Universal Robots URScript: faichun_snake3.script

def faichun_snake3():
  set_tool_communication(True, 1000000, 2, 1, 1.5, 3.5)
  set_tool_output_mode(0)
  set_tool_digital_output_mode(0, 1)
  set_tool_digital_output_mode(1, 1)
  set_tool_voltage(24)
  step_count_e741a7f4_0b30_46a8_b996_4636aff9ce90 = 0.0
  thread Step_Counter_Thread_bd4b55fe_d110_495a_a627_b98bcdc962aa():
    while (True):
      step_count_e741a7f4_0b30_46a8_b996_4636aff9ce90 = step_count_e741a7f4_0b30_46a8_b996_4636aff9ce90 + 1.0
      sync()
    end
  end
  run Step_Counter_Thread_bd4b55fe_d110_495a_a627_b98bcdc962aa()
  set_gravity([0.0, 0.0, 9.82])
  set_tcp(p[0.0,0.0,0.0,0.0,0.0,0.0])
  set_standard_analog_input_domain(0, 1)
  set_standard_analog_input_domain(1, 1)
  set_tool_analog_input_domain(0, 1)
  set_tool_analog_input_domain(1, 1)
  set_analog_outputdomain(0, 0)
  set_analog_outputdomain(1, 0)
  set_input_actions_to_default()
  set_safety_mode_transition_hardness(1)
  set_target_payload(1.070000, [0.002000, 0.003000, 0.057000], [0.001723, 0.001723, 0.001723, 0.000000, 0.000000, 0.000000])
  global B1empty=False
  global A2Empty=0
  global A1Empty=0
  global B2Empty=False
  global pallet_step=0
  global bright_box=0
  global Pallet_1_cnt=2
  global dark_boxes=0
  global Point_1=p[0.6913645118948067,-0.12399382748223003,0.49223711947071,-1.2983729986843258,1.1259514972191385,-1.2203503861141718]
  # begin: URCap Installation Node
  #   Source: External Control, 1.0.5, FZI Research Center for Information Technology
  #   Type: External Control
  # end: URCap Installation Node
  # begin: URCap Installation Node
  #   Source: OnRobot, 6.2.0, OnRobot A/S
  #   Type: OnRobot Setup
  sleep(1)
  if (False):
  end
  ON_CONN_SHIFT_BOOL = 64
  ON_CONN_SHIFT_INT = 24
  ON_CONN_SHIFT_FLOAT = 24
  ON_CONN_REG_SUM_BOOL = 0
  ON_CONN_REG_SUM_INT = 1
  ON_CONN_REG_SUM_FLOAT = 0
  ON_TOOL_SHIFT_BOOL = 64
  ON_TOOL_SHIFT_INT = 25
  ON_TOOL_SHIFT_FLOAT = 24
  ON_TOOL_SHIFT_BOOL_ARR = [64, 64, 64]
  ON_TOOL_SHIFT_INT_ARR = [25, 25, 25]
  ON_TOOL_SHIFT_FLOAT_ARR = [24, 24, 24]
  ON_TOOL_REG_SUM_BOOL = 0
  ON_TOOL_REG_SUM_INT = 0
  ON_TOOL_REG_SUM_FLOAT = 0
  ON_REGISTERS_SPEEDL_FLOAT = 0
  ON_REG_USE_TOOL = False
  ON_DI_SINGLE = 0
  ON_DI_PRIMARY = 1
  ON_DI_SECONDARY = 2
  ON_DI_DUAL = 3
  on_robot_type = 10
  on_robot_cycle = 2.0
  on_conn_ip = "localhost"
  on_tool_ip = "localhost"
  on_device_socket_port = 51234
  on_conn_xmlrpc = rpc_factory("xmlrpc", "http://localhost:41414")
  on_tool_xmlrpc = rpc_factory("xmlrpc", "http://localhost:41414")
  on_RPC = rpc_factory("xmlrpc", "http://127.0.0.1:31416")
  ON_DEBUG_LOG = False
  on_isMetric = True
  on_toolConnector = True
  on_ioqc = False
  on_dual = False
  on_computebox = False
  on_devices = 0
  on_gripper = [False, False, False]
  on_custom_tcp_id = "none"
  on_custom_tcp_enabled = False
  speedlTime = 0.001
  on_ft = False
  #======    OnRobot Globals    ======#

  ON_MATH_PI=3.141593
  ON_ZEROPOSE=p[0.0,0.0,0.0,0.0,0.0,0.0]
  ON_ZEROFRAME=p[0.0,0.0,0.0,0.0,0.0,0.0]
  ON_ZERO3D=[0.0,0.0,0.0]
  ON_ZERO6D=[0.0,0.0,0.0,0.0,0.0,0.0]
  ON_ZERO8D=[0.0,0.0,0.0,0.0,0.0,0.0,0.0,0.0]
  ON_FALSE3D=[False,False,False]
  ON_FALSE6D=[False,False,False,False,False,False]
  ON_FALSE8D=[False,False,False,False,False,False,False,False]
  global on_return=0
  on_speedL=ON_ZERO6D
  on_speedBase=ON_ZERO6D
  on_speedVect=ON_ZERO6D
  on_speedExtra=ON_ZERO6D
  on_speedCB=ON_ZERO6D
  on_speedGecko=ON_ZERO6D
  on_RTDE_error=0
  on_RTDE_tool_error=0
  on_dataProcess_thrd=0
  ON_DEVICE_ID_MISSING=0
  ON_INIT_WATCHDOG_HZ=5
  ON_INIT_TIMEOUT=2000
  on_robot_TCP_offset=ON_ZEROFRAME
  on_tcp_offset_actual=ON_ZEROFRAME
  on_cog_actual=ON_ZEROFRAME
  on_mass_actual=0.0
  on_robot_mount=[0.0,0.0]

  #======    End of OnRobot Globals    ======#
  #======    OnRobot Interface Messages    ======#

  on_devices_primary_log="OnRobot Devices"
  on_devices_secondary_log="OnRobot Secondary Device"
  on_program_halted="<br>Program halted."
  on_device_error_title="OnRobot - Device error"
  on_install_error="OnRobot Setup is not correct.<br>Check the status in the OnRobot Setup page in the Installation Tab.<br>Program halted."
  on_device_missing="No device connected.<br>Program halted."
  cb_device_missing="No OnRobot Compute Box connected.<br>Program halted."
  ft_device_missing="No OnRobot FT sensor or license detected.<br>Program halted."
  hex_device_missing="No HEX sensor connected.<br>Program halted."
  rg2ft_device_missing="No RG2-FT gripper connected.<br>Program halted."
  rg_device_missing="No RG gripper connected.<br>Program halted."
  vg_device_missing="No VG gripper connected.<br>Program halted."
  gg_device_missing="No Gecko Gripper connected.<br>Program halted."
  sg_device_missing="No Soft Gripper connected.<br>Program halted."
  tfg_device_missing="No 3FG gripper connected.<br>Program halted."
  sdr_device_missing="No OnRobot Sander connected.<br>Program halted."
  twofg_device_missing="No 2FG gripper connected.<br>Program halted."
  vgp_device_missing="No VGP gripper connected.<br>Program halted."
  mg_device_missing="No Magnetic Gripper connected.<br>Program halted."
  fgp_device_missing="No 2FGP20 Gripper connected.<br>Program halted."
  eyes_device_missing="No OnRobot Eyes connected.<br>Program halted."
  on_xmlrpc_start_ip="Connecting to OnRobot XML-RPC Server:"
  on_java_comm_error_textmsg_title="OnRobot - Communication error:"
  on_java_comm_controlsocket_open_error="Socket 'javaSocket' opening was unsuccessful."
  on_java_comm_error_title="OnRobot - Communication error"
  on_java_comm_socket_open_error="Establishing connection with the URCap was timed out.<br>Check the status in the OnRobot Setup page in the Installation Tab.<br>Program halted."
  on_rtde_feed_error_textmsg_title="OnRobot - RTDE error:"
  on_rtde_feed_error="RTDE feed error. OnRobot device count mismatch.<br>Program halted."
  on_rtde_feed_tool_error="Tool RTDE feed error. OnRobot device count mismatch.<br>Program halted."
  on_rtde_feed_open_error_textmsg="Socket 'rtdeFeed' opening was unsuccessful."
  on_rtde_feed_error_title="OnRobot - RTDE error"
  on_rtde_feed_count_error="Invalid RTDE offset setup detected. Please check RTDE Offsets at the OnRobot Setup page in the Installation Tab.<br>Program halted."
  on_rtde_feed_open_error="Establishing connection with the devices was timed out.<br>Ensure that the OnRobot devices are operational, and check the status in the OnRobot Setup page in the Installation Tab."

  #======    End of OnRobot Interface Messages    ======#
  #======    OnRobot Interface    ======#

  on_portopened_javaSocket=False
  on_rtde_feed_opened=False
  on_dataProcess_running=False
  def on_missing():
  popup(on_device_missing,title=on_device_error_title,error=True,blocking=False)
  halt
  end
  def cb_missing():
  popup(cb_device_missing,title=on_device_error_title,error=True,blocking=False)
  halt
  end
  def ft_missing():
  popup(ft_device_missing,title=on_device_error_title,error=True,blocking=False)
  halt
  end
  def hex_missing():
  popup(hex_device_missing,title=on_device_error_title,error=True,blocking=False)
  halt
  end
  def rg2ft_missing():
  popup(rg2ft_device_missing,title=on_device_error_title,error=True,blocking=False)
  halt
  end
  def rg_missing():
  popup(rg_device_missing,title=on_device_error_title,error=True,blocking=False)
  halt
  end
  def vg_missing():
  popup(vg_device_missing,title=on_device_error_title,error=True,blocking=False)
  halt
  end
  def gg_missing():
  popup(gg_device_missing,title=on_device_error_title,error=True,blocking=False)
  halt
  end
  def sg_missing():
  popup(sg_device_missing,title=on_device_error_title,error=True,blocking=False)
  halt
  end
  def tfg_missing():
  popup(tfg_device_missing,title=on_device_error_title,error=True,blocking=False)
  halt
  end
  def sdr_missing():
  popup(sdr_device_missing,title=on_device_error_title,error=True,blocking=False)
  halt
  end
  def twofg_missing():
  popup(twofg_device_missing,title=on_device_error_title,error=True,blocking=False)
  halt
  end
  def vgp_missing():
  popup(vgp_device_missing,title=on_device_error_title,error=True,blocking=False)
  halt
  end
  def mg_missing():
  popup(mg_device_missing,title=on_device_error_title,error=True,blocking=False)
  halt
  end
  def fgp_missing():
  popup(fgp_device_missing,title=on_device_error_title,error=True,blocking=False)
  halt
  end
  def eyes_missing():
  popup(eyes_device_missing,title=on_device_error_title,error=True,blocking=False)
  halt
  end
  def on_portclose_javaSocket():
  socket_close("javaSocket")
  on_portopened_javaSocket=False
  end
  def on_portopen_javaSocket():
  on_portclose_javaSocket()
  on_portopened_javaSocket=socket_open("127.0.0.1",44005,"javaSocket")
  if not on_portopened_javaSocket:
  textmsg(on_java_comm_error_textmsg_title,on_java_comm_controlsocket_open_error)
  popup(on_java_comm_socket_open_error,title=on_java_comm_error_title,error=True,blocking=False)
  halt
  end
  end
  on_conn_rtde_feed_name="rtdeFeedConn"
  on_tool_rtde_feed_name="rtdeFeedTool"
  def on_rtde_feed_close(rtdeFeedName):
  socket_close(rtdeFeedName)
  on_rtde_feed_opened=False
  end
  def on_rtde_feed_open(deviceIP,rtdeFeedName,regStart,regSum,regSpeedl):
  on_rtde_feed_close(rtdeFeedName)
  if((regStart[0]+regSum[0])>128)or((regStart[1]+regSum[1])>48)or((regStart[2]+regSum[2])>48):
  popup(on_rtde_feed_count_error,title=on_rtde_feed_error_title,error=True,blocking=False)
  textmsg(str_cat("RegStart: ",regStart),str_cat("  -  RegSum: ",regSum))
  halt
  end
  on_rtde_feed_opened=socket_open(deviceIP,on_device_socket_port,rtdeFeedName)
  if not on_rtde_feed_opened:
  on_rtde_feed_opened=socket_open(deviceIP,on_device_socket_port,rtdeFeedName)
  end
  if not on_rtde_feed_opened:
  textmsg(on_rtde_feed_error_textmsg_title,on_rtde_feed_open_error_textmsg)
  popup(on_rtde_feed_open_error,title=on_rtde_feed_error_title,error=True,blocking=False)
  halt
  end
  socket_send_int(regStart[0],rtdeFeedName)
  socket_send_int(regSum[0],rtdeFeedName)
  socket_send_int(regStart[1],rtdeFeedName)
  socket_send_int(regSum[1],rtdeFeedName)
  socket_send_int(regStart[2],rtdeFeedName)
  socket_send_int(regSum[2],rtdeFeedName)
  socket_send_int(regSpeedl,rtdeFeedName)
  socket_send_int(on_devices,rtdeFeedName)
  end
  def on_dataRead():
  enter_critical
  on_RTDE_error=read_input_integer_register(ON_CONN_SHIFT_INT)
  if(ON_REG_USE_TOOL):
  on_RTDE_tool_error=read_input_integer_register(ON_TOOL_SHIFT_INT_ARR[0])
  end
  exit_critical
  end
  def on_set_rtde_watchdog(updateHz=ON_INIT_WATCHDOG_HZ):
  local effect="stop"
  if(updateHz<1):
  effect="ignore"
  end
  watchdog_conn_reg_str=str_cat("input_int_register_",ON_CONN_SHIFT_INT)
  rtde_set_watchdog(watchdog_conn_reg_str,updateHz,effect)
  if(ON_REG_USE_TOOL):
  watchdog_tool_reg_str=str_cat("input_int_register_",ON_TOOL_SHIFT_INT_ARR[0])
  rtde_set_watchdog(watchdog_tool_reg_str,updateHz,effect)
  end
  if ON_DEBUG_LOG:
  local update_str=str_cat(" "+effect+" watchdog set to [Hz]: ",updateHz)
  textmsg(watchdog_conn_reg_str,update_str)
  if(ON_REG_USE_TOOL):
  local update_str=str_cat(" "+effect+" watchdog set to [Hz]: ",updateHz)
  textmsg(watchdog_tool_reg_str,update_str)
  end
  end
  end
  def on_speedCB_get():
  return[on_speedCB[0],on_speedCB[1],on_speedCB[2],on_speedCB[3],on_speedCB[4],on_speedCB[5]]
  end
  def on_speedGecko_get():
  local speedExtra=ON_ZERO6D
  if on_speedl_for_gecko:
  speedExtra=[on_speedGecko[0],on_speedGecko[1],on_speedGecko[2],on_speedGecko[3],on_speedGecko[4],on_speedGecko[5]]
  end
  return speedExtra
  end
  def on_speedGecko_set(speedGecko):
  on_speedGecko=[speedGecko[0],speedGecko[1],speedGecko[2],speedGecko[3],speedGecko[4],speedGecko[5]]
  end
  thread on_dataProcess_thread():
  if ON_DEBUG_LOG:
  textmsg("Starting on_dataRead thread")
  end
  local error=False
  on_dataProcess_running=True
  sync()
  while on_dataProcess_running:
  sync()
  on_dataRead()
  error=on_error((on_RTDE_error<0),on_rtde_feed_error,on_rtde_feed_error_title,error)
  error=on_error((ON_REG_USE_TOOL and(on_RTDE_tool_error<0)),on_rtde_feed_tool_error,on_rtde_feed_error_title,error)
  on_dataProcess_running=not error
  end
  if error:
  halt
  end
  if ON_DEBUG_LOG:
  textmsg("Stopping on_dataRead thread")
  end
  end
  thread on_set_watchdog_thread():
  sleep(2)
  on_set_rtde_watchdog(updateHz=ON_INIT_WATCHDOG_HZ)
  sleep(1/ON_INIT_WATCHDOG_HZ)
  on_dataProcess_running=False
  kill on_dataProcess_thrd
  end

  #======    End of OnRobot Interface    ======#
  #======    OnRobot QC Setup Tool Connector    ======#

  def tc_setup_tool():
  if ON_DEBUG_LOG:
  textmsg("QC Setup Tool Connector start...")
  end
  set_tool_voltage(24)

  set_tool_communication(True,1000000,2,1,1.5,3.5)

  if ON_DEBUG_LOG:
  textmsg("QC Setup Tool Connector end.")
  end
  end

  #======    End of OnRobot QC Setup Tool Connector    ======#
  #======    OnRobot TCP Messages    ======#

  on_tcp_log_msg_default="OnRobot: Robot TCP Offset set to:"
  on_tcp_log_msg_primary="OnRobot: Robot TCP Offset set to Primary:"
  on_tcp_log_msg_secondary="OnRobot: Robot TCP Offset set to Secondary:"

  #======    End of OnRobot TCP Messages    ======#
  #======    OnRobot TCP    ======#

  on_tcp_offset_actual=ON_ZEROFRAME
  on_tcp_offset_primary=ON_ZEROFRAME
  on_tcp_static_primary=ON_ZEROFRAME
  on_tcp_dynamic_primary=ON_ZEROFRAME
  on_tcp_adapters=ON_ZEROFRAME
  on_tcp_qc_primary=ON_ZEROFRAME
  on_tcp_base_primary=ON_ZEROFRAME
  on_tcp_gripper_static_primary=ON_ZEROFRAME
  on_tcp_workpiece_primary=ON_ZEROFRAME
  on_tcp_gripper_dynamic_primary=ON_ZEROFRAME
  on_tcp_gripper_primary=ON_ZEROFRAME
  on_tcp_offset_secondary=ON_ZEROFRAME
  on_tcp_static_secondary=ON_ZEROFRAME
  on_tcp_dynamic_secondary=ON_ZEROFRAME
  on_tcp_qc_secondary=ON_ZEROFRAME
  on_tcp_base_secondary=ON_ZEROFRAME
  on_tcp_gripper_static_secondary=ON_ZEROFRAME
  on_tcp_workpiece_secondary=ON_ZEROFRAME
  on_tcp_gripper_dynamic_secondary=ON_ZEROFRAME
  on_tcp_gripper_secondary=ON_ZEROFRAME
  on_tcp_custom_preset_assigned=False
  on_tcp_custom_preset=ON_ZEROFRAME
  def on_tcp_init_adapters():
  if ON_DEBUG_LOG:
  textmsg("TCP Init Adapters start..")
  end
  enter_critical
  on_tcp_adapters=ON_ZEROFRAME
  local adapterCount=length(on_tcp_adapters_array)
  local i=0
  while(i<adapterCount):
  on_tcp_adapters=pose_trans(on_tcp_adapters,on_tcp_adapters_array[i])
  i=i+1
  end
  exit_critical
  if ON_DEBUG_LOG:
  textmsg("TCP Init Adapters end.")
  end
  end
  def on_tcp_update_primary():
  if ON_DEBUG_LOG:
  textmsg("TCP Update Primary start..")
  end
  on_tcp_gripper_dynamic_primary=p[0.0, 0.0, 0.0, 0.0, 0.0, 0.0]
  enter_critical
  on_tcp_dynamic_primary=pose_trans(on_tcp_static_primary,on_tcp_gripper_dynamic_primary)
  on_tcp_offset_primary=pose_trans(on_tcp_dynamic_primary,on_tcp_workpiece_primary)
  exit_critical
  if ON_DEBUG_LOG:
  textmsg("TCP Update Primary end.")
  end
  end
  def on_tcp_init_primary():
  if ON_DEBUG_LOG:
  textmsg("TCP Init Primary start..")
  end
  enter_critical
  on_tcp_base_primary=pose_trans(on_tcp_adapters,on_tcp_qc_primary)
  on_tcp_static_primary=pose_trans(on_tcp_base_primary,on_tcp_gripper_static_primary)
  exit_critical
  on_tcp_update_primary()
  if ON_DEBUG_LOG:
  textmsg("TCP Init Primary end.")
  end
  end
  def on_tcp_offset_set(TCP_offset):
  if ON_DEBUG_LOG:
  textmsg("TCP Offset set started!")
  end
  on_tcp_offset_send(TCP_offset)
  if(on_follow_tcp):
  set_tcp(TCP_offset)
  end
  on_robot_TCP_offset=TCP_offset
  if ON_DEBUG_LOG:
  textmsg("TCP Offset set to: ",on_robot_TCP_offset)
  end
  end
  def on_tcp_offset_forced_set_actual(isPrimary=True):
  if(not on_follow_tcp):

  local tcp_log_msg=on_tcp_log_msg_default

  textmsg(tcp_log_msg,on_tcp_offset_actual)
  set_tcp(on_tcp_offset_actual)
  end
  end
  def on_tcp_update(isPrimary=True):
  on_tcp_update_primary()

  on_tcp_set_actual_to(isPrimary)
  end
  def on_tcp_set_actual_to(isPrimary=True):

  on_tcp_offset_actual=on_tcp_offset_primary
  if(on_follow_tcp):
  textmsg(on_tcp_log_msg_default,on_tcp_offset_actual)
  end

  on_tcp_active_is_primary=isPrimary
  on_tcp_offset_set(on_tcp_offset_actual)
  end
  def on_tcp_update_workpiece_primary(workpiece_offset):
  if ON_DEBUG_LOG:
  textmsg("TCP Update Tool Primary start..")
  end
  on_tcp_workpiece_primary=workpiece_offset
  on_tcp_update_primary()
  if ON_DEBUG_LOG:
  textmsg("TCP Update Tool Primary end.")
  end
  end
  def on_tcp_workpiece_rpy_get(xyz=[0.0,0.0,0.0],rpy=[0.0,0.0,0.0]):
  local rotvec=rpy2rotvec(rpy)
  local workpiece_offset=p[xyz[0],xyz[1],xyz[2],rotvec[0],rotvec[1],rotvec[2]]
  return workpiece_offset
  end

  def on_tcp_update_workpiece(workpiece_offset,tool_index=0):
  if ON_DEBUG_LOG:
  textmsg("TCP Update Tool start..")
  end
  if(tool_index!=ON_DI_SECONDARY):
  on_tcp_update_workpiece_primary(workpiece_offset)
  local isPrimary=True

  end
  on_tcp_set_actual_to(isPrimary)
  if ON_DEBUG_LOG:
  textmsg("TCP Update Tool end.")
  end
  end
  def on_get_tcp_for(tool_index):
  if tool_index==ON_DI_SECONDARY:
  local actual_tcp=on_tcp_static_secondary
  else:
  local actual_tcp=on_tcp_static_primary
  end
  return actual_tcp
  end
  def on_tcp_custom_unused():
  return ON_ZEROFRAME
  end
  def on_tcp_update_custom():
  if ON_DEBUG_LOG:
  textmsg("TCP Update Custom start..")
  end
  if(on_custom_tcp_enabled):
  on_tcp_custom_unused()
  on_tcp_custom_unused()
  on_tcp_custom_unused()
  on_tcp_custom_unused()

  end
  if ON_DEBUG_LOG:
  textmsg("TCP Update Custom end.")
  end
  end

  #======    End of OnRobot TCP    ======#
  #======    OnRobot Payload Messages    ======#

  on_mass_log_msg="OnRobot: Robot Payload Mass set to:"
  on_cog_log_msg="OnRobot: Robot Payload Center of Gravity set to:"

  #======    End of OnRobot Payload Messages    ======#
  #======    OnRobot Payload    ======#

  on_cog_actual=ON_ZEROFRAME
  on_mass_actual=0.0
  on_cog_primary=ON_ZEROFRAME
  on_cog_L1L2_primary=ON_ZEROFRAME
  on_mass_primary=0.0
  on_mass_L1L2_primary=0.0
  on_cog_adapters=ON_ZEROFRAME
  on_cog_qc_primary=ON_ZEROFRAME
  on_cog_base_primary=ON_ZEROFRAME
  on_cog_gripper_primary=ON_ZEROFRAME
  on_cog_workpiece_primary=ON_ZEROFRAME
  on_mass_adapters=0.0
  on_mass_qc_primary=0.0
  on_mass_base_primary=0.0
  on_mass_gripper_primary=0.0
  on_mass_workpiece_primary=0.0
  on_cog_secondary=ON_ZEROFRAME
  on_mass_secondary=0.0
  on_cog_gripper_secondary=ON_ZEROFRAME
  on_mass_gripper_secondary=0.0
  on_cog_workpiece_secondary=ON_ZEROFRAME
  on_mass_workpiece_secondary=0.0
  ON_LB2KG001=0.45359237/100
  def on_payload_init_adapters():
  if ON_DEBUG_LOG:
  textmsg("TCP Init Adapters start..")
  end
  enter_critical
  on_cog_adapters=ON_ZEROFRAME
  on_mass_adapters=0.0
  local massLAL0Ratio=0
  local adapterAbsCOG=ON_ZEROFRAME
  local tcp_adapter_offset=ON_ZEROFRAME
  local adapterCount=length(on_tcp_adapters_array)
  local i=0
  while(i<adapterCount):
  on_mass_adapters=on_mass_adapters+on_mass_adapters_array[i]
  if(on_mass_adapters<=0):
  massLAL0Ratio=0
  else:
  massLAL0Ratio=on_mass_adapters_array[i]/on_mass_adapters
  end
  adapterAbsCOG=pose_trans(tcp_adapter_offset,on_tcp_adapters_array[i])
  adapterAbsCOG=p[adapterAbsCOG[0],adapterAbsCOG[1],adapterAbsCOG[2],0.0,0.0,0.0]
  on_cog_adapters=interpolate_pose(on_cog_adapters,adapterAbsCOG,massLAL0Ratio)
  on_cog_adapters=p[on_cog_adapters[0],on_cog_adapters[1],on_cog_adapters[2],0.0,0.0,0.0]
  tcp_adapter_offset=pose_trans(tcp_adapter_offset,on_tcp_adapters_array[i])
  i=i+1
  sync()
  end
  exit_critical
  if ON_DEBUG_LOG:
  textmsg("TCP Init Adapters end.")
  end
  end
  def on_payload_update_primary():
  if ON_DEBUG_LOG:
  textmsg("Payload Update Primary start..")
  end
  enter_critical
  on_mass_primary=on_mass_L1L2_primary+on_mass_workpiece_primary
  local massL1L2L3Ratio=on_mass_workpiece_primary/on_mass_primary
  local workpieceAbsCOG=pose_trans(on_tcp_dynamic_primary,on_cog_workpiece_primary)
  workpieceAbsCOG=p[workpieceAbsCOG[0],workpieceAbsCOG[1],workpieceAbsCOG[2],0.0,0.0,0.0]
  on_cog_primary=interpolate_pose(on_cog_L1L2_primary,workpieceAbsCOG,massL1L2L3Ratio)
  on_cog_primary=p[on_cog_primary[0],on_cog_primary[1],on_cog_primary[2],0.0,0.0,0.0]
  exit_critical
  if ON_DEBUG_LOG:
  textmsg("Payload Update Primary end.")
  end
  end
  def on_payload_init_primary():
  if ON_DEBUG_LOG:
  textmsg("Payload Init Primary start..")
  end
  enter_critical
  on_mass_base_primary=on_mass_adapters+on_mass_qc_primary
  local massL0L1Ratio=on_mass_qc_primary/on_mass_base_primary
  on_mass_L1L2_primary=on_mass_base_primary+on_mass_gripper_primary
  local massL1L2Ratio=on_mass_gripper_primary/on_mass_L1L2_primary
  local qcAbsCOG=pose_trans(on_tcp_adapters,on_cog_qc_primary)
  qcAbsCOG=p[qcAbsCOG[0],qcAbsCOG[1],qcAbsCOG[2],0.0,0.0,0.0]
  on_cog_base_primary=interpolate_pose(on_cog_adapters,qcAbsCOG,massL0L1Ratio)
  on_cog_base_primary=p[on_cog_base_primary[0],on_cog_base_primary[1],on_cog_base_primary[2],0.0,0.0,0.0]
  local gripperAbsCOG=pose_trans(on_tcp_base_primary,on_cog_gripper_primary)
  gripperAbsCOG=p[gripperAbsCOG[0],gripperAbsCOG[1],gripperAbsCOG[2],0.0,0.0,0.0]
  on_cog_L1L2_primary=interpolate_pose(on_cog_base_primary,gripperAbsCOG,massL1L2Ratio)
  on_cog_L1L2_primary=p[on_cog_L1L2_primary[0],on_cog_L1L2_primary[1],on_cog_L1L2_primary[2],0.0,0.0,0.0]
  exit_critical
  on_payload_update_primary()
  if ON_DEBUG_LOG:
  textmsg("Payload Init Primary end.")
  end
  end
  def on_payload_update():
  on_payload_update_primary()

  on_mass_actual =on_mass_primary
  on_cog_actual=on_cog_primary

  on_payload_set_actual()
  end
  def on_payload_set_actual():

  on_mass_actual =on_mass_primary
  on_cog_actual=on_cog_primary

  local CoG=[on_cog_actual[0],on_cog_actual[1],on_cog_actual[2]]
  on_payload_set(on_mass_actual,CoG)
  end
  def on_payload_update_workpiece_primary(workpiece_mass=0,workpiece_cog=[0.0,0.0,0.0]):
  if ON_DEBUG_LOG:
  textmsg("Payload Update Workpiece Primary start..")
  end
  on_cog_workpiece_primary=p[workpiece_cog[0],workpiece_cog[1],workpiece_cog[2],0.0,0.0,0.0]
  on_mass_workpiece_primary=workpiece_mass
  on_payload_update_primary()
  if ON_DEBUG_LOG:
  textmsg("Payload Update Workpiece Primary end.")
  end
  end
  def on_payload_set(mass,CoG):
  if ON_DEBUG_LOG:
  textmsg("Payload set started!")
  end
  local center_of_gravity=[CoG[0],CoG[1],CoG[2]]
  on_payload_send(center_of_gravity,mass)
  if(on_isMetric):
  local roundedMass=floor(mass*100+0.5)/100
  else:
  local roundedMass=floor(mass/ON_LB2KG001+0.5)*ON_LB2KG001
  end
  set_payload(roundedMass,center_of_gravity)
  on_mass_actual=roundedMass
  on_cog_actual=p[CoG[0],CoG[1],CoG[2],0.0,0.0,0.0]
  if ON_DEBUG_LOG:
  textmsg("Payload mass, CoG set to: ",str_cat(str_cat(mass,", "),CoG))
  end
  end

  def on_payload_update_secondary():
  end
  def on_payload_init_secondary():
  end

  def on_payload_update_workpiece(workpiece_mass,workpiece_cog=[0.0,0.0,0.0],tool_index=0):
  if ON_DEBUG_LOG:
  textmsg("Payload Update Workpiece start..")
  end
  if(tool_index!=ON_DI_SECONDARY):
  on_cog_workpiece_primary=p[workpiece_cog[0],workpiece_cog[1],workpiece_cog[2],0.0,0.0,0.0]
  on_mass_workpiece_primary=workpiece_mass
  else:
  on_cog_workpiece_secondary=p[workpiece_cog[0],workpiece_cog[1],workpiece_cog[2],0.0,0.0,0.0]
  on_mass_workpiece_secondary=workpiece_mass
  end
  on_payload_update()
  if ON_DEBUG_LOG:
  textmsg("Payload Update Workpiece end.")
  end
  end
  def on_payload_get_cog2tcp_workpiece(tool_index=0):
  if(tool_index!=ON_DI_SECONDARY):
  local cog_tool=[on_tcp_workpiece_primary[0],on_tcp_workpiece_primary[1],on_tcp_workpiece_primary[2]]
  else:
  local cog_tool=[on_tcp_workpiece_secondary[0],on_tcp_workpiece_secondary[1],on_tcp_workpiece_secondary[2]]
  end
  return cog_tool
  end

  #======    End of OnRobot Payload    ======#
  #======    OnRobot QC TCP    ======#

  onrobotmini=0

  def on_tcp_offset_send(TCP_offset):
  on_robot_TCP_offset=TCP_offset
  end
  def on_payload_send(CoG,mass):
  on_robot_payload_cog=CoG
  on_robot_payload_mass=mass
  end


  #======    End of OnRobot QC TCP    ======#
  #======    OnRobot  Speedl    ======#

  on_speedl_thread_handler=0
  on_speedl_is_enabled=False
  on_speedl_is_running=False
  on_speedl_acc=0.0
  ft_speedl_hg_caranteen_reached=False
  ft_speedl_hg_caranteen_safemode=False
  on_speedl_for_ftcontrol=False
  on_speedl_for_move=False
  on_speedl_for_handguide=False
  on_speedl_for_insertpart=False
  on_speedl_for_depthcompensation=False
  on_speedl_for_center=False
  on_speedl_for_gecko=False
  on_speedl_acc=10000.0
  on_speedl_acc_to_zero=3.0
  ON_SPEEDL_FTCONTROL=1
  ON_SPEEDL_HANDGUIDE=2
  ON_SPEEDL_TRAJECTORY=3
  ON_SPEEDL_MOVE=ON_SPEEDL_TRAJECTORY
  ON_SPEEDL_INSERTPART=4
  ON_SPEEDL_DEPTHCOMP=5
  ON_SPEEDL_CENTER=6
  ON_SPEEDL_GECKO=7
  def on_wait_ms(time_ms):
  local sync_time=ceil(norm(time_ms/2.0))
  while(sync_time>0):
  sync_time=sync_time-1
  sync()
  end
  end
  def on_error(status_flag,message,title,stop_var=False):
  if(status_flag):
  popup(message,title=title,error=True,blocking=False)
  stop_var=True
  end
  return stop_var
  end
  def on_warning(status_flag,message,title,isPopupNeeded=False,is_shown=False):
  if(status_flag):
  if(not is_shown):
  if(isPopupNeeded):
  popup(message,title=title,warning=True,blocking=False)
  else:
  textmsg(title+": ",message)
  end
  is_shown=True
  end
  else:
  is_shown=False
  end
  return is_shown
  end
  def on_speedl_add_extra(speedBase,speedExtra):
  speedSum=ON_ZERO6D
  speedBaseP=p[speedBase[0],speedBase[1],speedBase[2],speedBase[3],speedBase[4],speedBase[5]]
  speedExtraP=p[speedExtra[0],speedExtra[1],speedExtra[2],speedExtra[3],speedExtra[4],speedExtra[5]]
  speedSumP=pose_add(speedExtraP,speedBaseP)
  speedSum=[speedSumP[0],speedSumP[1],speedSumP[2],speedSumP[3],speedSumP[4],speedSumP[5]]
  return speedSum
  end

  thread on_speedl_thread():
  if ON_DEBUG_LOG:
  textmsg("Speedl thread started..")
  end
  enter_critical
  on_speedl_is_running=True
  on_speedl_is_enabled=True
  exit_critical
  on_speedL=ON_ZERO6D
  on_speedL_last=ON_ZERO6D

  while on_speedl_is_running:
  on_speedBase=on_speedCB_get()
  on_speedL=on_speedBase


  if on_speedl_is_enabled:
  if(on_speedL==ON_ZERO6D):
  on_speedL=[on_speedL_last[0]/100,on_speedL_last[1]/100,on_speedL_last[2]/100,on_speedL_last[3]/100,on_speedL_last[4]/100,on_speedL_last[5]/100]
  end
  speedl(on_speedL,a=on_speedl_acc,t=speedlTime)
  else:
  speedl(ON_ZERO6D,a=on_speedl_acc_to_zero,t=speedlTime)
  end
  on_speedL_last=on_speedL
  end

  on_speedL=ON_ZERO6D
  if ON_DEBUG_LOG:
  textmsg("Speedl thread ended.")
  end
  end
  def on_speedl_integer_get():
  local speedl_integer=binary_list_to_integer([on_speedl_for_ftcontrol,on_speedl_for_handguide,on_speedl_for_move,on_speedl_for_insertpart,on_speedl_for_depthcompensation,on_speedl_for_center,on_speedl_for_gecko])
  return speedl_integer
  end
  def on_speedl_start_for(speedl_id):
  if(speedl_id==ON_SPEEDL_FTCONTROL):
  on_speedl_for_ftcontrol=True
  elif(speedl_id==ON_SPEEDL_HANDGUIDE):
  on_speedl_for_handguide=True
  elif(speedl_id==ON_SPEEDL_TRAJECTORY):
  on_speedl_for_move=True
  elif(speedl_id==ON_SPEEDL_INSERTPART):
  on_speedl_for_insertpart=True
  elif(speedl_id==ON_SPEEDL_DEPTHCOMP):
  on_speedl_for_depthcompensation=True
  elif(speedl_id==ON_SPEEDL_CENTER):
  on_speedl_for_center=True
  elif(speedl_id==ON_SPEEDL_GECKO):
  on_speedl_for_gecko=True
  else:
  textmsg("Unknown Start speedl ID received: ",speedl_id)
  end
  local speedl_integer=on_speedl_integer_get()
  if not(speedl_integer==0):
  if not on_speedl_is_running:
  on_speedl_thread_handler=run on_speedl_thread()
  end
  end
  return on_speedl_is_running
  end
  def on_speedl_stop_for(speedl_id,brake=10,brakeRot=10):
  if(speedl_id==ON_SPEEDL_FTCONTROL):
  on_speedl_for_ftcontrol=False
  elif(speedl_id==ON_SPEEDL_HANDGUIDE):
  on_speedl_for_handguide=False
  elif(speedl_id==ON_SPEEDL_TRAJECTORY):
  on_speedl_for_move=False
  elif(speedl_id==ON_SPEEDL_INSERTPART):
  on_speedl_for_insertpart=False
  elif(speedl_id==ON_SPEEDL_DEPTHCOMP):
  on_speedl_for_depthcompensation=False
  elif(speedl_id==ON_SPEEDL_CENTER):
  on_speedl_for_center=False
  elif(speedl_id==ON_SPEEDL_GECKO):
  on_speedl_for_gecko=False
  on_speedGecko_set(ON_ZERO6D)
  else:
  textmsg("Unknown Stop speedl ID received: ",speedl_id)
  end
  local speedl_integer=on_speedl_integer_get()
  if(speedl_integer==0):
  if(on_speedl_is_running):
  kill on_speedl_thread_handler
  enter_critical
  on_speedl_is_running=False
  exit_critical

  end
  if ON_DEBUG_LOG:
  textmsg("Speedl thread stopped")
  end
  stopl(brake,brakeRot)
  end
  return on_speedl_is_running
  end
  def on_speedl_pause():
  on_speedl_is_enabled=False
  return on_speedl_integer_get()
  end
  def on_speedl_resume():
  on_speedl_is_enabled=True
  return on_speedl_integer_get()
  end

  #======    End of OnRobot  Speedl    ======#
  textmsg(on_devices_primary_log, ": Quick Changer + QC Tool Side + [0.0, 0.0, 0.0, 0.0, 0.0, 0.0]")
  on_follow_tcp = False
  on_tcp_active_is_primary = True
  on_tcp_adapters_array = []
  on_cog_adapters_array = []
  on_mass_adapters_array = []
  on_tcp_qc_primary = p[0.0, 0.0, 0.0136, 0.0, 0.0, 0.0]
  on_cog_qc_primary = p[0.0, 0.0, 0.004, 0.0, 0.0, 0.0]
  on_mass_qc_primary = 0.06
  on_tcp_gripper_static_primary = p[0.0, 0.0, 0.017, 0.0, 0.0, 0.0]
  on_cog_gripper_primary = p[0.0, 0.0, 0.002, 0.0, 0.0, 0.0]
  on_mass_gripper_primary = 0.14
  on_tcp_workpiece_primary = p[0.0, 0.0, 0.0, 0.0, 0.0, 0.0]
  on_cog_workpiece_primary = p[0.0, 0.0, 0.0, 0.0, 0.0, 0.0]
  on_mass_workpiece_primary = 0.0
  #======    OnRobot Run    ======#

  on_portopen_javaSocket()
  sync()
  textmsg(on_xmlrpc_start_ip,on_conn_ip)
  if(ON_REG_USE_TOOL):
  on_regStart_conn=[ON_CONN_SHIFT_BOOL,ON_CONN_SHIFT_INT,ON_CONN_SHIFT_FLOAT]
  on_regSum_conn=[ON_CONN_REG_SUM_BOOL,ON_CONN_REG_SUM_INT,ON_CONN_REG_SUM_FLOAT]
  on_rtde_feed_open(on_conn_ip,on_conn_rtde_feed_name,on_regStart_conn,on_regSum_conn,ON_REGISTERS_SPEEDL_FLOAT)
  sync()
  textmsg(on_xmlrpc_start_ip,on_tool_ip)
  on_regStart_tool=[ON_TOOL_SHIFT_BOOL,ON_TOOL_SHIFT_INT,ON_TOOL_SHIFT_FLOAT]
  on_regSum_tool=[ON_TOOL_REG_SUM_BOOL,ON_TOOL_REG_SUM_INT,ON_TOOL_REG_SUM_FLOAT]
  on_rtde_feed_open(on_tool_ip,on_tool_rtde_feed_name,on_regStart_tool,on_regSum_tool,0)
  sync()
  else:
  on_regStart_conn=[ON_CONN_SHIFT_BOOL,ON_CONN_SHIFT_INT,ON_CONN_SHIFT_FLOAT]
  on_regSum_conn=[ON_CONN_REG_SUM_BOOL,ON_CONN_REG_SUM_INT,ON_CONN_REG_SUM_FLOAT]
  on_rtde_feed_open(on_conn_ip,on_conn_rtde_feed_name,on_regStart_conn,on_regSum_conn,ON_REGISTERS_SPEEDL_FLOAT)
  sync()
  end
  on_set_rtde_watchdog(updateHz=0.2)
  sync()
  on_dataProcess_thrd=run on_dataProcess_thread()
  sync()
  on_tcp_init_adapters()
  on_payload_init_adapters()
  on_tcp_init_primary()
  on_payload_init_primary()

  on_tcp_update_custom()
  on_tcp_set_actual_to(on_tcp_active_is_primary)
  if(on_follow_tcp):
  on_payload_set_actual()
  end
  on_watchdog_thrd=run on_set_watchdog_thread()
  sync()
  def done_waiting_for_init(device_name,product_code,tool_index=0):
  textmsg(str_cat(device_name,str_cat(str_cat("[",tool_index),"]: ")),product_code)
  end

  #======    End of OnRobot Run    ======#
  #======    OnRobot QC Start    ======#

  if(on_toolConnector):
  tc_setup_tool()
  end
  sync()

  #======    End of OnRobot QC Start    ======#
  # end: URCap Installation Node
  $ 1 "Robot Program"
  $ 2 "Script: FaiChun_9 Jan_11_2_t1_2.script"
  def Machining1():
    # Default parameters:
    global speed_ms = 0.05
    global speed_rads = 0.75
    global accel_mss = 3
    global accel_radss = 1.2
    global blend_radius_m = 0.0003

    # Add subprograms here
    # Start of main program
    # Program generated by RoboDK v5.6.8 for UR10e on 17/01/2025 17:23:54
    # Using nominal kinematics.
    blend_radius_m = 0.0003
    speed_ms = 0.05
    # set_reference(p[0.340000, -0.238000, 0.001500, 0.000000, 0.000000, 0.000000])
    set_tcp(p[0.000000, 0.000000, 0.252000, 0.000000, 0.000000, 0.000000])
    # Show Tool
    movej([0.145114, -1.397514, -2.446396, -0.868479, 1.570796, 1.715910],accel_radss,speed_rads,0,blend_radius_m)
    movel([0.145114, -1.450226, -2.476289, -0.785874, 1.570796, 1.715910],accel_mss,speed_ms,0,blend_radius_m)
    #SetTool1
    #M_RunCode6
    #SetRPM60000
    speed_ms = 0.05
    #M_RunCode3
    movel([0.145114, -1.473196, -2.487384, -0.751808, 1.570796, 1.715910],accel_mss,speed_ms,0,blend_radius_m)
    speed_ms = 0.003
    movel([0.145114, -1.479129, -2.490086, -0.743174, 1.570796, 1.715910],accel_mss,speed_ms,0,blend_radius_m)
    speed_ms = 0.05
    movel([-0.131626, -1.561533, -2.414291, -0.736565, 1.570796, 1.439170],accel_mss,speed_ms,0,blend_radius_m)
    movel([-0.177704, -1.331249, -2.600139, -0.781001, 1.570796, 1.393092],accel_mss,speed_ms,0,blend_radius_m)
    movel([0.204954, -1.166991, -2.688242, -0.857156, 1.570796, 1.775750],accel_mss,speed_ms,0,blend_radius_m)
    movel([0.145114, -1.479129, -2.490086, -0.743174, 1.570796, 1.715910],accel_mss,speed_ms,0,blend_radius_m)
    speed_ms = 0.003
    movel([0.145114, -1.473196, -2.487384, -0.751808, 1.570796, 1.715910],accel_mss,speed_ms,0,blend_radius_m)
    speed_ms = 0.05
    movel([0.145114, -1.450226, -2.476289, -0.785874, 1.570796, 1.715910],accel_mss,speed_ms,0,blend_radius_m)
    #M_RunCode9
    movel([0.141001, -1.443521, -2.481739, -0.787129, 1.570796, 1.711798],accel_mss,speed_ms,0,blend_radius_m)
    #M_RunCode3
    movel([0.141001, -1.466629, -2.492914, -0.752846, 1.570796, 1.711798],accel_mss,speed_ms,0,blend_radius_m)
    speed_ms = 0.003
    movel([0.141001, -1.472599, -2.495635, -0.744154, 1.570796, 1.711798],accel_mss,speed_ms,0,blend_radius_m)
    speed_ms = 0.012
    movel([0.136639, -1.473494, -2.494879, -0.744016, 1.570796, 1.707435],accel_mss,speed_ms,0,blend_radius_m)
    movel([0.136042, -1.477254, -2.491686, -0.743449, 1.570796, 1.706838],accel_mss,speed_ms,0,blend_radius_m)
    movel([0.129615, -1.478592, -2.490545, -0.743252, 1.570796, 1.700411],accel_mss,speed_ms,0,blend_radius_m)
    movel([0.130181, -1.474842, -2.493736, -0.743810, 1.570796, 1.700977],accel_mss,speed_ms,0,blend_radius_m)
    movel([0.127919, -1.475323, -2.493329, -0.743738, 1.570796, 1.698716],accel_mss,speed_ms,0,blend_radius_m)
    movel([0.127361, -1.479068, -2.490138, -0.743183, 1.570796, 1.698157],accel_mss,speed_ms,0,blend_radius_m)
    movel([0.121982, -1.480222, -2.489150, -0.743016, 1.570796, 1.692778],accel_mss,speed_ms,0,blend_radius_m)
    movel([0.120939, -1.480446, -2.488958, -0.742984, 1.570796, 1.691735],accel_mss,speed_ms,0,blend_radius_m)
    movel([0.121724, -1.474915, -2.493675, -0.743799, 1.570796, 1.692520],accel_mss,speed_ms,0,blend_radius_m)
    movel([0.126089, -1.473968, -2.494478, -0.743944, 1.570796, 1.696886],accel_mss,speed_ms,0,blend_radius_m)
    movel([0.126378, -1.472012, -2.496131, -0.744246, 1.570796, 1.697174],accel_mss,speed_ms,0,blend_radius_m)
    movel([0.119733, -1.473463, -2.494905, -0.744021, 1.570796, 1.690529],accel_mss,speed_ms,0,blend_radius_m)
    movel([0.118690, -1.480938, -2.488537, -0.742914, 1.570796, 1.689486],accel_mss,speed_ms,0,blend_radius_m)
    movel([0.117647, -1.481168, -2.488339, -0.742882, 1.570796, 1.688443],accel_mss,speed_ms,0,blend_radius_m)
    speed_ms = 0.02
    movel([0.002864, -1.511155, -2.461903, -0.739330, 1.570796, 1.573661],accel_mss,speed_ms,0,blend_radius_m)
    movel([-0.108286, -1.549104, -2.426413, -0.736872, 1.570796, 1.462510],accel_mss,speed_ms,0,blend_radius_m)
    speed_ms = 0.012
    movel([-0.109170, -1.542784, -2.432482, -0.737123, 1.570796, 1.461626],accel_mss,speed_ms,0,blend_radius_m)
    movel([-0.115268, -1.545135, -2.430232, -0.737022, 1.570796, 1.455529],accel_mss,speed_ms,0,blend_radius_m)
    movel([-0.115029, -1.546770, -2.428662, -0.736957, 1.570796, 1.455767],accel_mss,speed_ms,0,blend_radius_m)
    movel([-0.111023, -1.545226, -2.430145, -0.737018, 1.570796, 1.459773],accel_mss,speed_ms,0,blend_radius_m)
    movel([-0.110365, -1.549892, -2.425652, -0.736845, 1.570796, 1.460431],accel_mss,speed_ms,0,blend_radius_m)
    movel([-0.111325, -1.550258, -2.425297, -0.736833, 1.570796, 1.459472],accel_mss,speed_ms,0,blend_radius_m)
    movel([-0.116260, -1.552156, -2.423459, -0.736774, 1.570796, 1.454536],accel_mss,speed_ms,0,blend_radius_m)
    movel([-0.116726, -1.549025, -2.426489, -0.736875, 1.570796, 1.454070],accel_mss,speed_ms,0,blend_radius_m)
    movel([-0.118795, -1.549827, -2.425715, -0.736847, 1.570796, 1.452001],accel_mss,speed_ms,0,blend_radius_m)
    movel([-0.118321, -1.552953, -2.422685, -0.736751, 1.570796, 1.452475],accel_mss,speed_ms,0,blend_radius_m)
    movel([-0.124187, -1.555237, -2.420462, -0.736690, 1.570796, 1.446609],accel_mss,speed_ms,0,blend_radius_m)
    movel([-0.124683, -1.552129, -2.423485, -0.736775, 1.570796, 1.446114],accel_mss,speed_ms,0,blend_radius_m)
    movel([-0.128648, -1.553694, -2.421965, -0.736730, 1.570796, 1.442148],accel_mss,speed_ms,0,blend_radius_m)
    movel([-0.129411, -1.549091, -2.426425, -0.736873, 1.570796, 1.441385],accel_mss,speed_ms,0,blend_radius_m)
    movel([-0.125425, -1.547510, -2.427949, -0.736929, 1.570796, 1.445371],accel_mss,speed_ms,0,blend_radius_m)
    movel([-0.125687, -1.545886, -2.429511, -0.736992, 1.570796, 1.445109],accel_mss,speed_ms,0,blend_radius_m)
    movel([-0.129681, -1.547471, -2.427987, -0.736931, 1.570796, 1.441115],accel_mss,speed_ms,0,blend_radius_m)
    movel([-0.130331, -1.543596, -2.431706, -0.737087, 1.570796, 1.440465],accel_mss,speed_ms,0,blend_radius_m)
    movel([-0.130456, -1.542840, -2.432429, -0.737120, 1.570796, 1.440341],accel_mss,speed_ms,0,blend_radius_m)
    movel([-0.124505, -1.540465, -2.434693, -0.737231, 1.570796, 1.446291],accel_mss,speed_ms,0,blend_radius_m)
    movel([-0.124003, -1.543613, -2.431690, -0.737086, 1.570796, 1.446793],accel_mss,speed_ms,0,blend_radius_m)
    movel([-0.121918, -1.542790, -2.432476, -0.737122, 1.570796, 1.448878],accel_mss,speed_ms,0,blend_radius_m)
    movel([-0.122672, -1.537996, -2.437038, -0.737355, 1.570796, 1.448124],accel_mss,speed_ms,0,blend_radius_m)
    movel([-0.130730, -1.541209, -2.433985, -0.737195, 1.570796, 1.440067],accel_mss,speed_ms,0,blend_radius_m)
    movel([-0.146735, -1.452072, -2.512652, -0.747665, 1.570796, 1.424062],accel_mss,speed_ms,0,blend_radius_m)
    speed_ms = 0.02
    movel([-0.166789, -1.353893, -2.585329, -0.773167, 1.570796, 1.404008],accel_mss,speed_ms,0,blend_radius_m)
    movel([-0.166990, -1.352958, -2.585955, -0.773476, 1.570796, 1.403806],accel_mss,speed_ms,0,blend_radius_m)
    speed_ms = 0.012
    movel([-0.156896, -1.347760, -2.589410, -0.775219, 1.570796, 1.413900],accel_mss,speed_ms,0,blend_radius_m)
    movel([-0.158123, -1.341762, -2.593351, -0.777277, 1.570796, 1.412674],accel_mss,speed_ms,0,blend_radius_m)
    movel([-0.160766, -1.343128, -2.592457, -0.776804, 1.570796, 1.410031],accel_mss,speed_ms,0,blend_radius_m)
    movel([-0.159947, -1.347068, -2.589867, -0.775454, 1.570796, 1.410849],accel_mss,speed_ms,0,blend_radius_m)
    movel([-0.167424, -1.350932, -2.587305, -0.774151, 1.570796, 1.403372],accel_mss,speed_ms,0,blend_radius_m)
    movel([-0.167629, -1.349998, -2.587927, -0.774464, 1.570796, 1.403168],accel_mss,speed_ms,0,blend_radius_m)
    movel([-0.168693, -1.345153, -2.591129, -0.776107, 1.570796, 1.402103],accel_mss,speed_ms,0,blend_radius_m)
    movel([-0.163615, -1.342502, -2.592867, -0.777020, 1.570796, 1.407181],accel_mss,speed_ms,0,blend_radius_m)
    movel([-0.164053, -1.340454, -2.594203, -0.777732, 1.570796, 1.406744],accel_mss,speed_ms,0,blend_radius_m)
    movel([-0.169143, -1.343118, -2.592464, -0.776807, 1.570796, 1.401654],accel_mss,speed_ms,0,blend_radius_m)
    movel([-0.170437, -1.337285, -2.596260, -0.778844, 1.570796, 1.400359],accel_mss,speed_ms,0,blend_radius_m)
    movel([-0.165313, -1.334580, -2.598005, -0.779805, 1.570796, 1.405484],accel_mss,speed_ms,0,blend_radius_m)
    movel([-0.166173, -1.330591, -2.600559, -0.781239, 1.570796, 1.404623],accel_mss,speed_ms,0,blend_radius_m)
    movel([-0.158508, -1.326548, -2.603127, -0.782714, 1.570796, 1.412289],accel_mss,speed_ms,0,blend_radius_m)
    movel([-0.157682, -1.330578, -2.600567, -0.781243, 1.570796, 1.413114],accel_mss,speed_ms,0,blend_radius_m)
    movel([-0.154998, -1.329179, -2.601459, -0.781752, 1.570796, 1.415798],accel_mss,speed_ms,0,blend_radius_m)
    movel([-0.155811, -1.325133, -2.604020, -0.783236, 1.570796, 1.414985],accel_mss,speed_ms,0,blend_radius_m)
    movel([-0.148083, -1.321101, -2.606551, -0.784737, 1.570796, 1.422714],accel_mss,speed_ms,0,blend_radius_m)
    movel([-0.146935, -1.327148, -2.602747, -0.782494, 1.570796, 1.423861],accel_mss,speed_ms,0,blend_radius_m)
    movel([-0.152123, -1.329828, -2.601046, -0.781516, 1.570796, 1.418673],accel_mss,speed_ms,0,blend_radius_m)
    movel([-0.151712, -1.331924, -2.599708, -0.780757, 1.570796, 1.419084],accel_mss,speed_ms,0,blend_radius_m)
    movel([-0.143841, -1.327877, -2.602285, -0.782227, 1.570796, 1.426955],accel_mss,speed_ms,0,blend_radius_m)
    movel([-0.145364, -1.319691, -2.607431, -0.785267, 1.570796, 1.425432],accel_mss,speed_ms,0,blend_radius_m)
    movel([0.003920, -1.248574, -2.648506, -0.815310, 1.570796, 1.574716],accel_mss,speed_ms,0,blend_radius_m)
    speed_ms = 0.02
    movel([0.165154, -1.186625, -2.679348, -0.846417, 1.570796, 1.735951],accel_mss,speed_ms,0,blend_radius_m)
    movel([0.163152, -1.198149, -2.673935, -0.840305, 1.570796, 1.733948],accel_mss,speed_ms,0,blend_radius_m)
    speed_ms = 0.012
    movel([0.172319, -1.195184, -2.675341, -0.841863, 1.570796, 1.743115],accel_mss,speed_ms,0,blend_radius_m)
    movel([0.172866, -1.192193, -2.676750, -0.843445, 1.570796, 1.743662],accel_mss,speed_ms,0,blend_radius_m)
    movel([0.166811, -1.194153, -2.675828, -0.842408, 1.570796, 1.737608],accel_mss,speed_ms,0,blend_radius_m)
    movel([0.168335, -1.185580, -2.679831, -0.846978, 1.570796, 1.739131],accel_mss,speed_ms,0,blend_radius_m)
    movel([0.169806, -1.185096, -2.680055, -0.847238, 1.570796, 1.740602],accel_mss,speed_ms,0,blend_radius_m)
    movel([0.177391, -1.182622, -2.681194, -0.848573, 1.570796, 1.748187],accel_mss,speed_ms,0,blend_radius_m)
    movel([0.176304, -1.188464, -2.678494, -0.845432, 1.570796, 1.747100],accel_mss,speed_ms,0,blend_radius_m)
    movel([0.179460, -1.187457, -2.678962, -0.845971, 1.570796, 1.750256],accel_mss,speed_ms,0,blend_radius_m)
    movel([0.180574, -1.181595, -2.681665, -0.849129, 1.570796, 1.751371],accel_mss,speed_ms,0,blend_radius_m)
    movel([0.189651, -1.178707, -2.682983, -0.850699, 1.570796, 1.760447],accel_mss,speed_ms,0,blend_radius_m)
    movel([0.188481, -1.184611, -2.680279, -0.847499, 1.570796, 1.759277],accel_mss,speed_ms,0,blend_radius_m)
    movel([0.194577, -1.182720, -2.681149, -0.848520, 1.570796, 1.765374],accel_mss,speed_ms,0,blend_radius_m)
    movel([0.192814, -1.191401, -2.677122, -0.843866, 1.570796, 1.763610],accel_mss,speed_ms,0,blend_radius_m)
    movel([0.186775, -1.193250, -2.676254, -0.842885, 1.570796, 1.757572],accel_mss,speed_ms,0,blend_radius_m)
    movel([0.186185, -1.196251, -2.674837, -0.841302, 1.570796, 1.756982],accel_mss,speed_ms,0,blend_radius_m)
    movel([0.192203, -1.194418, -2.675703, -0.842268, 1.570796, 1.762999],accel_mss,speed_ms,0,blend_radius_m)
    movel([0.190761, -1.201563, -2.672304, -0.838522, 1.570796, 1.761557],accel_mss,speed_ms,0,blend_radius_m)
    movel([0.190484, -1.202941, -2.671643, -0.837806, 1.570796, 1.761280],accel_mss,speed_ms,0,blend_radius_m)
    movel([0.181657, -1.205609, -2.670355, -0.836426, 1.570796, 1.752453],accel_mss,speed_ms,0,blend_radius_m)
    movel([0.182758, -1.199906, -2.673098, -0.839385, 1.570796, 1.753554],accel_mss,speed_ms,0,blend_radius_m)
    movel([0.179644, -1.200868, -2.672637, -0.838884, 1.570796, 1.750441],accel_mss,speed_ms,0,blend_radius_m)
    movel([0.178007, -1.209492, -2.668466, -0.834430, 1.570796, 1.748803],accel_mss,speed_ms,0,blend_radius_m)
    movel([0.189888, -1.205903, -2.670212, -0.836273, 1.570796, 1.760685],accel_mss,speed_ms,0,blend_radius_m)
    speed_ms = 0.02
    movel([0.163402, -1.343756, -2.592046, -0.776587, 1.570796, 1.734198],accel_mss,speed_ms,0,blend_radius_m)
    movel([0.143535, -1.457310, -2.508372, -0.746708, 1.570796, 1.714331],accel_mss,speed_ms,0,blend_radius_m)
    speed_ms = 0.012
    movel([0.134639, -1.459191, -2.506824, -0.746374, 1.570796, 1.705436],accel_mss,speed_ms,0,blend_radius_m)
    movel([0.133732, -1.465007, -2.502005, -0.745377, 1.570796, 1.704528],accel_mss,speed_ms,0,blend_radius_m)
    movel([0.136023, -1.464522, -2.502409, -0.745459, 1.570796, 1.706819],accel_mss,speed_ms,0,blend_radius_m)
    movel([0.136629, -1.460695, -2.505582, -0.746111, 1.570796, 1.707425],accel_mss,speed_ms,0,blend_radius_m)
    movel([0.143192, -1.459319, -2.506719, -0.746352, 1.570796, 1.713988],accel_mss,speed_ms,0,blend_radius_m)
    movel([0.143038, -1.460245, -2.505954, -0.746190, 1.570796, 1.713835],accel_mss,speed_ms,0,blend_radius_m)
    movel([0.142251, -1.464999, -2.502011, -0.745379, 1.570796, 1.713048],accel_mss,speed_ms,0,blend_radius_m)
    movel([0.137849, -1.465911, -2.501251, -0.745227, 1.570796, 1.708646],accel_mss,speed_ms,0,blend_radius_m)
    movel([0.137533, -1.467886, -2.499600, -0.744903, 1.570796, 1.708330],accel_mss,speed_ms,0,blend_radius_m)
    movel([0.141927, -1.466979, -2.500359, -0.745051, 1.570796, 1.712723],accel_mss,speed_ms,0,blend_radius_m)
    movel([0.141001, -1.472599, -2.495635, -0.744154, 1.570796, 1.711798],accel_mss,speed_ms,0,blend_radius_m)
    speed_ms = 0.003
    movel([0.141001, -1.466629, -2.492914, -0.752846, 1.570796, 1.711798],accel_mss,speed_ms,0,blend_radius_m)
    speed_ms = 0.05
    movel([0.141001, -1.443521, -2.481739, -0.787129, 1.570796, 1.711798],accel_mss,speed_ms,0,blend_radius_m)
    #M_RunCode9
    movel([-0.095971, -1.320143, -2.570643, -0.821603, 1.570796, 1.474826],accel_mss,speed_ms,0,blend_radius_m)
    #M_RunCode3
    # num 0 inside
    movel([-0.095971, -1.345583, -2.583353, -0.783454, 1.570796, 1.474826],accel_mss,speed_ms,0,blend_radius_m)
    speed_ms = 0.003
    movel([-0.095971, -1.352203, -2.586459, -0.773727, 1.570796, 1.474826],accel_mss,speed_ms,0,blend_radius_m)
    speed_ms = 0.015
    movel([-0.101060, -1.358991, -2.581897, -0.771501, 1.570796, 1.469736],accel_mss,speed_ms,0,blend_radius_m)
    movel([-0.105019, -1.363609, -2.578758, -0.770023, 1.570796, 1.465778],accel_mss,speed_ms,0,blend_radius_m)
    movel([-0.106639, -1.365123, -2.577722, -0.769544, 1.570796, 1.464157],accel_mss,speed_ms,0,blend_radius_m)
    movel([-0.108096, -1.366111, -2.577044, -0.769234, 1.570796, 1.462701],accel_mss,speed_ms,0,blend_radius_m)
    movel([-0.109388, -1.366578, -2.576723, -0.769088, 1.570796, 1.461409],accel_mss,speed_ms,0,blend_radius_m)
    movel([-0.110520, -1.366524, -2.576760, -0.769105, 1.570796, 1.460276],accel_mss,speed_ms,0,blend_radius_m)
    movel([-0.111321, -1.366002, -2.577119, -0.769268, 1.570796, 1.459475],accel_mss,speed_ms,0,blend_radius_m)
    movel([-0.111616, -1.365061, -2.577764, -0.769564, 1.570796, 1.459180],accel_mss,speed_ms,0,blend_radius_m)
    movel([-0.111403, -1.363700, -2.578696, -0.769994, 1.570796, 1.459393],accel_mss,speed_ms,0,blend_radius_m)
    movel([-0.110683, -1.361913, -2.579914, -0.770562, 1.570796, 1.460113],accel_mss,speed_ms,0,blend_radius_m)
    movel([-0.107823, -1.356944, -2.583280, -0.772165, 1.570796, 1.462973],accel_mss,speed_ms,0,blend_radius_m)
    movel([-0.103126, -1.350010, -2.587919, -0.774460, 1.570796, 1.467671],accel_mss,speed_ms,0,blend_radius_m)
    movel([-0.097993, -1.343109, -2.592470, -0.776810, 1.570796, 1.472803],accel_mss,speed_ms,0,blend_radius_m)
    movel([-0.093909, -1.338331, -2.595583, -0.778476, 1.570796, 1.476888],accel_mss,speed_ms,0,blend_radius_m)
    movel([-0.092221, -1.336752, -2.596604, -0.779033, 1.570796, 1.478576],accel_mss,speed_ms,0,blend_radius_m)
    movel([-0.090706, -1.335718, -2.597272, -0.779399, 1.570796, 1.480090],accel_mss,speed_ms,0,blend_radius_m)
    movel([-0.089366, -1.335233, -2.597584, -0.779572, 1.570796, 1.481430],accel_mss,speed_ms,0,blend_radius_m)
    movel([-0.088203, -1.335298, -2.597543, -0.779549, 1.570796, 1.482593],accel_mss,speed_ms,0,blend_radius_m)
    movel([-0.087396, -1.335857, -2.597182, -0.779350, 1.570796, 1.483400],accel_mss,speed_ms,0,blend_radius_m)
    movel([-0.087120, -1.336850, -2.596541, -0.778998, 1.570796, 1.483676],accel_mss,speed_ms,0,blend_radius_m)
    movel([-0.087378, -1.338279, -2.595616, -0.778494, 1.570796, 1.483418],accel_mss,speed_ms,0,blend_radius_m)
    movel([-0.088162, -1.340134, -2.594412, -0.777843, 1.570796, 1.482634],accel_mss,speed_ms,0,blend_radius_m)
    movel([-0.091172, -1.345231, -2.591077, -0.776081, 1.570796, 1.479624],accel_mss,speed_ms,0,blend_radius_m)
    movel([-0.095971, -1.352203, -2.586459, -0.773727, 1.570796, 1.474826],accel_mss,speed_ms,0,blend_radius_m)
    speed_ms = 0.003
    movel([-0.095971, -1.345583, -2.583353, -0.783454, 1.570796, 1.474826],accel_mss,speed_ms,0,blend_radius_m)
    speed_ms = 0.05
    movel([-0.095971, -1.320143, -2.570643, -0.821603, 1.570796, 1.474826],accel_mss,speed_ms,0,blend_radius_m)
    #M_RunCode9
    movel([-0.088305, -1.322635, -2.569052, -0.820702, 1.570796, 1.482491],accel_mss,speed_ms,0,blend_radius_m)
    #M_RunCode3
    #num 0 outside
    movel([-0.088305, -1.348033, -2.581729, -0.782626, 1.570796, 1.482491],accel_mss,speed_ms,0,blend_radius_m)
    speed_ms = 0.003
    movel([-0.088305, -1.354642, -2.584827, -0.772920, 1.570796, 1.482491],accel_mss,speed_ms,0,blend_radius_m)
    speed_ms = 0.015
    movel([-0.090204, -1.357095, -2.583178, -0.772116, 1.570796, 1.480592],accel_mss,speed_ms,0,blend_radius_m)
    movel([-0.092146, -1.359299, -2.581689, -0.771401, 1.570796, 1.478650],accel_mss,speed_ms,0,blend_radius_m)
    movel([-0.094134, -1.361259, -2.580359, -0.770771, 1.570796, 1.476662],accel_mss,speed_ms,0,blend_radius_m)
    movel([-0.096168, -1.362974, -2.579191, -0.770224, 1.570796, 1.474629],accel_mss,speed_ms,0,blend_radius_m)
    movel([-0.098207, -1.364435, -2.578193, -0.769761, 1.570796, 1.472589],accel_mss,speed_ms,0,blend_radius_m)
    movel([-0.100213, -1.365632, -2.577372, -0.769384, 1.570796, 1.470584],accel_mss,speed_ms,0,blend_radius_m)
    movel([-0.102186, -1.366569, -2.576729, -0.769091, 1.570796, 1.468610],accel_mss,speed_ms,0,blend_radius_m)
    movel([-0.104128, -1.367242, -2.576266, -0.768881, 1.570796, 1.466669],accel_mss,speed_ms,0,blend_radius_m)
    movel([-0.106011, -1.367658, -2.575980, -0.768751, 1.570796, 1.464785],accel_mss,speed_ms,0,blend_radius_m)
    movel([-0.107803, -1.367820, -2.575868, -0.768701, 1.570796, 1.462993],accel_mss,speed_ms,0,blend_radius_m)
    movel([-0.109510, -1.367730, -2.575930, -0.768729, 1.570796, 1.461286],accel_mss,speed_ms,0,blend_radius_m)
    movel([-0.111131, -1.367388, -2.576166, -0.768835, 1.570796, 1.459665],accel_mss,speed_ms,0,blend_radius_m)
    movel([-0.112591, -1.366814, -2.576561, -0.769014, 1.570796, 1.458205],accel_mss,speed_ms,0,blend_radius_m)
    movel([-0.113810, -1.366033, -2.577098, -0.769259, 1.570796, 1.456987],accel_mss,speed_ms,0,blend_radius_m)
    movel([-0.114791, -1.365044, -2.577776, -0.769569, 1.570796, 1.456006],accel_mss,speed_ms,0,blend_radius_m)
    movel([-0.115530, -1.363841, -2.578599, -0.769949, 1.570796, 1.455266],accel_mss,speed_ms,0,blend_radius_m)
    movel([-0.116005, -1.362439, -2.579556, -0.770394, 1.570796, 1.454792],accel_mss,speed_ms,0,blend_radius_m)
    movel([-0.116190, -1.360849, -2.580638, -0.770902, 1.570796, 1.454606],accel_mss,speed_ms,0,blend_radius_m)
    movel([-0.116085, -1.359067, -2.581846, -0.771476, 1.570796, 1.454711],accel_mss,speed_ms,0,blend_radius_m)
    movel([-0.115685, -1.357091, -2.583180, -0.772117, 1.570796, 1.455111],accel_mss,speed_ms,0,blend_radius_m)
    movel([-0.114980, -1.354950, -2.584621, -0.772819, 1.570796, 1.455816],accel_mss,speed_ms,0,blend_radius_m)
    movel([-0.113953, -1.352671, -2.586146, -0.773572, 1.570796, 1.456843],accel_mss,speed_ms,0,blend_radius_m)
    movel([-0.112603, -1.350256, -2.587755, -0.774378, 1.570796, 1.458193],accel_mss,speed_ms,0,blend_radius_m)
    movel([-0.110928, -1.347704, -2.589447, -0.775238, 1.570796, 1.459868],accel_mss,speed_ms,0,blend_radius_m)
    movel([-0.109051, -1.345192, -2.591103, -0.776094, 1.570796, 1.461745],accel_mss,speed_ms,0,blend_radius_m)
    movel([-0.107107, -1.342916, -2.592596, -0.776877, 1.570796, 1.463689],accel_mss,speed_ms,0,blend_radius_m)
    movel([-0.105094, -1.340873, -2.593931, -0.777586, 1.570796, 1.465702],accel_mss,speed_ms,0,blend_radius_m)
    movel([-0.103017, -1.339070, -2.595103, -0.778216, 1.570796, 1.467780],accel_mss,speed_ms,0,blend_radius_m)
    movel([-0.100919, -1.337525, -2.596105, -0.778759, 1.570796, 1.469878],accel_mss,speed_ms,0,blend_radius_m)
    movel([-0.098849, -1.336258, -2.596923, -0.779208, 1.570796, 1.471947],accel_mss,speed_ms,0,blend_radius_m)
    movel([-0.096809, -1.335267, -2.597562, -0.779560, 1.570796, 1.473987],accel_mss,speed_ms,0,blend_radius_m)
    movel([-0.094800, -1.334558, -2.598018, -0.779812, 1.570796, 1.475997],accel_mss,speed_ms,0,blend_radius_m)
    movel([-0.092856, -1.334126, -2.598296, -0.779966, 1.570796, 1.477940],accel_mss,speed_ms,0,blend_radius_m)
    movel([-0.091005, -1.333963, -2.598401, -0.780025, 1.570796, 1.479791],accel_mss,speed_ms,0,blend_radius_m)
    movel([-0.089247, -1.334068, -2.598334, -0.779987, 1.570796, 1.481550],accel_mss,speed_ms,0,blend_radius_m)
    movel([-0.087589, -1.334445, -2.598091, -0.779853, 1.570796, 1.483208],accel_mss,speed_ms,0,blend_radius_m)
    movel([-0.086106, -1.335067, -2.597691, -0.779631, 1.570796, 1.484690],accel_mss,speed_ms,0,blend_radius_m)
    movel([-0.084880, -1.335904, -2.597152, -0.779333, 1.570796, 1.485916],accel_mss,speed_ms,0,blend_radius_m)
    movel([-0.083910, -1.336959, -2.596471, -0.778959, 1.570796, 1.486886],accel_mss,speed_ms,0,blend_radius_m)
    movel([-0.083195, -1.338228, -2.595649, -0.778512, 1.570796, 1.487601],accel_mss,speed_ms,0,blend_radius_m)
    movel([-0.082761, -1.339697, -2.594696, -0.777996, 1.570796, 1.488035],accel_mss,speed_ms,0,blend_radius_m)
    movel([-0.082632, -1.341356, -2.593615, -0.777417, 1.570796, 1.488165],accel_mss,speed_ms,0,blend_radius_m)
    movel([-0.082808, -1.343205, -2.592407, -0.776777, 1.570796, 1.487989],accel_mss,speed_ms,0,blend_radius_m)
    movel([-0.083285, -1.345236, -2.591074, -0.776079, 1.570796, 1.487512],accel_mss,speed_ms,0,blend_radius_m)
    movel([-0.084070, -1.347416, -2.589637, -0.775336, 1.570796, 1.486727],accel_mss,speed_ms,0,blend_radius_m)
    movel([-0.085171, -1.349713, -2.588116, -0.774560, 1.570796, 1.485626],accel_mss,speed_ms,0,blend_radius_m)
    movel([-0.086583, -1.352122, -2.586513, -0.773754, 1.570796, 1.484213],accel_mss,speed_ms,0,blend_radius_m)
    movel([-0.088305, -1.354642, -2.584827, -0.772920, 1.570796, 1.482491],accel_mss,speed_ms,0,blend_radius_m)
    speed_ms = 0.003
    movel([-0.088305, -1.348033, -2.581729, -0.782626, 1.570796, 1.482491],accel_mss,speed_ms,0,blend_radius_m)
    speed_ms = 0.05
    movel([-0.088305, -1.322635, -2.569052, -0.820702, 1.570796, 1.482491],accel_mss,speed_ms,0,blend_radius_m)
    #M_RunCode9
    movel([-0.118832, -1.321958, -2.569485, -0.820946, 1.570796, 1.451964],accel_mss,speed_ms,0,blend_radius_m)
    #M_RunCode3
    movel([-0.118832, -1.347368, -2.582171, -0.782850, 1.570796, 1.451964],accel_mss,speed_ms,0,blend_radius_m)
    speed_ms = 0.003
    movel([-0.118832, -1.353979, -2.585271, -0.773138, 1.570796, 1.451964],accel_mss,speed_ms,0,blend_radius_m)
    speed_ms = 0.02
    movel([-0.124934, -1.362775, -2.579327, -0.770287, 1.570796, 1.445862],accel_mss,speed_ms,0,blend_radius_m)
    movel([-0.148632, -1.356620, -2.583498, -0.772271, 1.570796, 1.422164],accel_mss,speed_ms,0,blend_radius_m)
    movel([-0.148043, -1.355734, -2.584094, -0.772561, 1.570796, 1.422754],accel_mss,speed_ms,0,blend_radius_m)
    movel([-0.146262, -1.353538, -2.585567, -0.773284, 1.570796, 1.424534],accel_mss,speed_ms,0,blend_radius_m)
    movel([-0.143953, -1.351516, -2.586917, -0.773956, 1.570796, 1.426844],accel_mss,speed_ms,0,blend_radius_m)
    movel([-0.141315, -1.349690, -2.588131, -0.774568, 1.570796, 1.429481],accel_mss,speed_ms,0,blend_radius_m)
    movel([-0.138559, -1.348086, -2.589194, -0.775109, 1.570796, 1.432238],accel_mss,speed_ms,0,blend_radius_m)
    movel([-0.130967, -1.344319, -2.591676, -0.776393, 1.570796, 1.439829],accel_mss,speed_ms,0,blend_radius_m)
    movel([-0.123880, -1.340890, -2.593919, -0.777580, 1.570796, 1.446916],accel_mss,speed_ms,0,blend_radius_m)
    movel([-0.121261, -1.339412, -2.594881, -0.778096, 1.570796, 1.449535],accel_mss,speed_ms,0,blend_radius_m)
    movel([-0.118795, -1.337754, -2.595956, -0.778678, 1.570796, 1.452001],accel_mss,speed_ms,0,blend_radius_m)
    movel([-0.116656, -1.335945, -2.597125, -0.779319, 1.570796, 1.454140],accel_mss,speed_ms,0,blend_radius_m)
    movel([-0.115017, -1.334007, -2.598373, -0.780009, 1.570796, 1.455779],accel_mss,speed_ms,0,blend_radius_m)
    movel([-0.113700, -1.331542, -2.599952, -0.780895, 1.570796, 1.457096],accel_mss,speed_ms,0,blend_radius_m)
    movel([-0.113452, -1.330481, -2.600629, -0.781279, 1.570796, 1.457345],accel_mss,speed_ms,0,blend_radius_m)
    movel([-0.113477, -1.329535, -2.601232, -0.781622, 1.570796, 1.457320],accel_mss,speed_ms,0,blend_radius_m)
    movel([-0.114162, -1.328078, -2.602158, -0.782154, 1.570796, 1.456635],accel_mss,speed_ms,0,blend_radius_m)
    movel([-0.115566, -1.327268, -2.602671, -0.782450, 1.570796, 1.455230],accel_mss,speed_ms,0,blend_radius_m)
    movel([-0.116775, -1.327100, -2.602777, -0.782511, 1.570796, 1.454022],accel_mss,speed_ms,0,blend_radius_m)
    movel([-0.117884, -1.327287, -2.602659, -0.782443, 1.570796, 1.452913],accel_mss,speed_ms,0,blend_radius_m)
    movel([-0.118818, -1.327765, -2.602356, -0.782268, 1.570796, 1.451978],accel_mss,speed_ms,0,blend_radius_m)
    movel([-0.119500, -1.328465, -2.601912, -0.782012, 1.570796, 1.451297],accel_mss,speed_ms,0,blend_radius_m)
    movel([-0.119848, -1.329672, -2.601145, -0.781572, 1.570796, 1.450949],accel_mss,speed_ms,0,blend_radius_m)
    movel([-0.120081, -1.330839, -2.600401, -0.781149, 1.570796, 1.450715],accel_mss,speed_ms,0,blend_radius_m)
    movel([-0.120851, -1.332269, -2.599487, -0.780633, 1.570796, 1.449945],accel_mss,speed_ms,0,blend_radius_m)
    movel([-0.122252, -1.333823, -2.598491, -0.780075, 1.570796, 1.448544],accel_mss,speed_ms,0,blend_radius_m)
    movel([-0.123926, -1.334807, -2.597858, -0.779723, 1.570796, 1.446870],accel_mss,speed_ms,0,blend_radius_m)
    movel([-0.125677, -1.335229, -2.597587, -0.779573, 1.570796, 1.445119],accel_mss,speed_ms,0,blend_radius_m)
    movel([-0.127302, -1.335096, -2.597672, -0.779620, 1.570796, 1.443494],accel_mss,speed_ms,0,blend_radius_m)
    movel([-0.128587, -1.334465, -2.598078, -0.779846, 1.570796, 1.442210],accel_mss,speed_ms,0,blend_radius_m)
    movel([-0.129320, -1.333388, -2.598770, -0.780231, 1.570796, 1.441477],accel_mss,speed_ms,0,blend_radius_m)
    movel([-0.129352, -1.331950, -2.599691, -0.780748, 1.570796, 1.441444],accel_mss,speed_ms,0,blend_radius_m)
    movel([-0.128528, -1.330238, -2.600784, -0.781367, 1.570796, 1.442268],accel_mss,speed_ms,0,blend_radius_m)
    movel([-0.127385, -1.328836, -2.601677, -0.781877, 1.570796, 1.443412],accel_mss,speed_ms,0,blend_radius_m)
    movel([-0.126030, -1.327695, -2.602400, -0.782293, 1.570796, 1.444766],accel_mss,speed_ms,0,blend_radius_m)
    movel([-0.124463, -1.326815, -2.602958, -0.782616, 1.570796, 1.446334],accel_mss,speed_ms,0,blend_radius_m)
    movel([-0.122683, -1.326203, -2.603345, -0.782841, 1.570796, 1.448113],accel_mss,speed_ms,0,blend_radius_m)
    movel([-0.120785, -1.325853, -2.603565, -0.782970, 1.570796, 1.450011],accel_mss,speed_ms,0,blend_radius_m)
    movel([-0.118858, -1.325758, -2.603626, -0.783005, 1.570796, 1.451938],accel_mss,speed_ms,0,blend_radius_m)
    movel([-0.114926, -1.326342, -2.603257, -0.782790, 1.570796, 1.455870],accel_mss,speed_ms,0,blend_radius_m)
    movel([-0.112673, -1.327135, -2.602755, -0.782499, 1.570796, 1.458123],accel_mss,speed_ms,0,blend_radius_m)
    movel([-0.110749, -1.328180, -2.602093, -0.782116, 1.570796, 1.460048],accel_mss,speed_ms,0,blend_radius_m)
    movel([-0.109155, -1.329474, -2.601271, -0.781644, 1.570796, 1.461641],accel_mss,speed_ms,0,blend_radius_m)
    movel([-0.107892, -1.331014, -2.600289, -0.781086, 1.570796, 1.462904],accel_mss,speed_ms,0,blend_radius_m)
    movel([-0.107162, -1.332798, -2.599148, -0.780443, 1.570796, 1.463634],accel_mss,speed_ms,0,blend_radius_m)
    movel([-0.107176, -1.334831, -2.597843, -0.779715, 1.570796, 1.463620],accel_mss,speed_ms,0,blend_radius_m)
    movel([-0.107927, -1.337107, -2.596375, -0.778907, 1.570796, 1.462869],accel_mss,speed_ms,0,blend_radius_m)
    movel([-0.109406, -1.339620, -2.594746, -0.778023, 1.570796, 1.461391],accel_mss,speed_ms,0,blend_radius_m)
    movel([-0.111183, -1.341801, -2.593325, -0.777263, 1.570796, 1.459613],accel_mss,speed_ms,0,blend_radius_m)
    movel([-0.113261, -1.343698, -2.592084, -0.776607, 1.570796, 1.457535],accel_mss,speed_ms,0,blend_radius_m)
    movel([-0.115524, -1.345335, -2.591009, -0.776045, 1.570796, 1.455272],accel_mss,speed_ms,0,blend_radius_m)
    movel([-0.117852, -1.346735, -2.590087, -0.775567, 1.570796, 1.452944],accel_mss,speed_ms,0,blend_radius_m)
    movel([-0.123738, -1.349638, -2.588166, -0.774585, 1.570796, 1.447059],accel_mss,speed_ms,0,blend_radius_m)
    movel([-0.129266, -1.352407, -2.586322, -0.773659, 1.570796, 1.441530],accel_mss,speed_ms,0,blend_radius_m)
    movel([-0.131364, -1.353673, -2.585476, -0.773239, 1.570796, 1.439432],accel_mss,speed_ms,0,blend_radius_m)
    movel([-0.133365, -1.355125, -2.584503, -0.772761, 1.570796, 1.437431],accel_mss,speed_ms,0,blend_radius_m)
    movel([-0.135159, -1.356768, -2.583398, -0.772223, 1.570796, 1.435638],accel_mss,speed_ms,0,blend_radius_m)
    movel([-0.136628, -1.358602, -2.582161, -0.771626, 1.570796, 1.434168],accel_mss,speed_ms,0,blend_radius_m)
    movel([-0.135740, -1.358833, -2.582004, -0.771552, 1.570796, 1.435057],accel_mss,speed_ms,0,blend_radius_m)
    movel([-0.133192, -1.359344, -2.581658, -0.771387, 1.570796, 1.437605],accel_mss,speed_ms,0,blend_radius_m)
    movel([-0.130761, -1.359508, -2.581548, -0.771334, 1.570796, 1.440035],accel_mss,speed_ms,0,blend_radius_m)
    movel([-0.128449, -1.359327, -2.581670, -0.771392, 1.570796, 1.442347],accel_mss,speed_ms,0,blend_radius_m)
    movel([-0.126248, -1.358795, -2.582030, -0.771564, 1.570796, 1.444548],accel_mss,speed_ms,0,blend_radius_m)
    movel([-0.124179, -1.357967, -2.582590, -0.771832, 1.570796, 1.446617],accel_mss,speed_ms,0,blend_radius_m)
    movel([-0.122254, -1.356890, -2.583316, -0.772183, 1.570796, 1.448542],accel_mss,speed_ms,0,blend_radius_m)
    movel([-0.120474, -1.355562, -2.584210, -0.772617, 1.570796, 1.450322],accel_mss,speed_ms,0,blend_radius_m)
    movel([-0.118832, -1.353979, -2.585271, -0.773138, 1.570796, 1.451964],accel_mss,speed_ms,0,blend_radius_m)
    speed_ms = 0.003
    movel([-0.118832, -1.347368, -2.582171, -0.782850, 1.570796, 1.451964],accel_mss,speed_ms,0,blend_radius_m)
    speed_ms = 0.05
    movel([-0.118832, -1.321958, -2.569485, -0.820946, 1.570796, 1.451964],accel_mss,speed_ms,0,blend_radius_m)
    #M_RunCode9
    movel([0.073358, -1.418214, -2.501717, -0.792458, 1.570796, 1.644154],accel_mss,speed_ms,0,blend_radius_m)
    #M_RunCode3
    movel([0.073358, -1.441837, -2.513195, -0.757357, 1.570796, 1.644154],accel_mss,speed_ms,0,blend_radius_m)
    speed_ms = 0.003
    movel([0.073358, -1.447948, -2.515992, -0.748448, 1.570796, 1.644154],accel_mss,speed_ms,0,blend_radius_m)
    speed_ms = 0.02
    movel([0.075270, -1.446294, -2.517325, -0.748770, 1.570796, 1.646066],accel_mss,speed_ms,0,blend_radius_m)
    movel([0.077554, -1.444921, -2.518428, -0.749040, 1.570796, 1.648350],accel_mss,speed_ms,0,blend_radius_m)
    movel([0.080047, -1.443807, -2.519321, -0.749261, 1.570796, 1.650843],accel_mss,speed_ms,0,blend_radius_m)
    movel([0.082577, -1.442932, -2.520021, -0.749436, 1.570796, 1.653374],accel_mss,speed_ms,0,blend_radius_m)
    movel([0.089381, -1.441132, -2.521457, -0.749800, 1.570796, 1.660178],accel_mss,speed_ms,0,blend_radius_m)
    movel([0.095696, -1.439540, -2.522724, -0.750126, 1.570796, 1.666492],accel_mss,speed_ms,0,blend_radius_m)
    movel([0.098074, -1.438760, -2.523343, -0.750287, 1.570796, 1.668870],accel_mss,speed_ms,0,blend_radius_m)
    movel([0.100372, -1.437779, -2.524119, -0.750490, 1.570796, 1.671168],accel_mss,speed_ms,0,blend_radius_m)
    movel([0.102449, -1.436586, -2.525063, -0.750740, 1.570796, 1.673245],accel_mss,speed_ms,0,blend_radius_m)
    movel([0.104165, -1.435162, -2.526185, -0.751041, 1.570796, 1.674961],accel_mss,speed_ms,0,blend_radius_m)
    movel([0.105751, -1.433181, -2.527743, -0.751465, 1.570796, 1.676547],accel_mss,speed_ms,0,blend_radius_m)
    movel([0.106187, -1.432257, -2.528467, -0.751665, 1.570796, 1.676983],accel_mss,speed_ms,0,blend_radius_m)
    movel([0.106384, -1.431377, -2.529156, -0.751856, 1.570796, 1.677181],accel_mss,speed_ms,0,blend_radius_m)
    movel([0.106189, -1.429873, -2.530330, -0.752186, 1.570796, 1.676986],accel_mss,speed_ms,0,blend_radius_m)
    movel([0.105289, -1.428805, -2.531162, -0.752422, 1.570796, 1.676086],accel_mss,speed_ms,0,blend_radius_m)
    movel([0.104393, -1.428371, -2.531499, -0.752519, 1.570796, 1.675190],accel_mss,speed_ms,0,blend_radius_m)
    movel([0.103490, -1.428293, -2.531560, -0.752536, 1.570796, 1.674286],accel_mss,speed_ms,0,blend_radius_m)
    movel([0.102658, -1.428519, -2.531384, -0.752486, 1.570796, 1.673455],accel_mss,speed_ms,0,blend_radius_m)
    movel([0.101969, -1.429012, -2.531001, -0.752376, 1.570796, 1.672765],accel_mss,speed_ms,0,blend_radius_m)
    movel([0.101420, -1.430050, -2.530192, -0.752147, 1.570796, 1.672216],accel_mss,speed_ms,0,blend_radius_m)
    movel([0.100969, -1.431080, -2.529388, -0.751921, 1.570796, 1.671765],accel_mss,speed_ms,0,blend_radius_m)
    movel([0.100039, -1.432229, -2.528489, -0.751671, 1.570796, 1.670835],accel_mss,speed_ms,0,blend_radius_m)
    movel([0.098595, -1.433352, -2.527609, -0.751428, 1.570796, 1.669391],accel_mss,speed_ms,0,blend_radius_m)
    movel([0.097067, -1.433883, -2.527192, -0.751314, 1.570796, 1.667864],accel_mss,speed_ms,0,blend_radius_m)
    movel([0.095608, -1.433877, -2.527196, -0.751315, 1.570796, 1.666404],accel_mss,speed_ms,0,blend_radius_m)
    movel([0.094378, -1.433385, -2.527583, -0.751421, 1.570796, 1.665174],accel_mss,speed_ms,0,blend_radius_m)
    movel([0.093528, -1.432503, -2.528274, -0.751611, 1.570796, 1.664324],accel_mss,speed_ms,0,blend_radius_m)
    movel([0.093210, -1.431334, -2.529189, -0.751866, 1.570796, 1.664006],accel_mss,speed_ms,0,blend_radius_m)
    movel([0.093521, -1.429992, -2.530237, -0.752160, 1.570796, 1.664317],accel_mss,speed_ms,0,blend_radius_m)
    movel([0.094560, -1.428589, -2.531329, -0.752470, 1.570796, 1.665357],accel_mss,speed_ms,0,blend_radius_m)
    movel([0.095773, -1.427547, -2.532139, -0.752703, 1.570796, 1.666569],accel_mss,speed_ms,0,blend_radius_m)
    movel([0.097091, -1.426799, -2.532719, -0.752871, 1.570796, 1.667888],accel_mss,speed_ms,0,blend_radius_m)
    movel([0.098510, -1.426345, -2.533071, -0.752973, 1.570796, 1.669306],accel_mss,speed_ms,0,blend_radius_m)
    movel([0.100028, -1.426187, -2.533193, -0.753009, 1.570796, 1.670824],accel_mss,speed_ms,0,blend_radius_m)
    movel([0.101578, -1.426298, -2.533108, -0.752984, 1.570796, 1.672374],accel_mss,speed_ms,0,blend_radius_m)
    movel([0.103090, -1.426654, -2.532832, -0.752903, 1.570796, 1.673886],accel_mss,speed_ms,0,blend_radius_m)
    movel([0.105998, -1.428092, -2.531716, -0.752581, 1.570796, 1.676795],accel_mss,speed_ms,0,blend_radius_m)
    movel([0.107557, -1.429342, -2.530744, -0.752303, 1.570796, 1.678354],accel_mss,speed_ms,0,blend_radius_m)
    movel([0.108806, -1.430745, -2.529650, -0.751994, 1.570796, 1.679602],accel_mss,speed_ms,0,blend_radius_m)
    movel([0.109743, -1.432300, -2.528433, -0.751655, 1.570796, 1.680539],accel_mss,speed_ms,0,blend_radius_m)
    movel([0.110369, -1.434007, -2.527094, -0.751288, 1.570796, 1.681165],accel_mss,speed_ms,0,blend_radius_m)
    movel([0.110526, -1.435818, -2.525669, -0.750902, 1.570796, 1.681322],accel_mss,speed_ms,0,blend_radius_m)
    movel([0.110053, -1.437690, -2.524190, -0.750509, 1.570796, 1.680850],accel_mss,speed_ms,0,blend_radius_m)
    movel([0.108957, -1.439621, -2.522659, -0.750109, 1.570796, 1.679754],accel_mss,speed_ms,0,blend_radius_m)
    movel([0.107237, -1.441611, -2.521075, -0.749702, 1.570796, 1.678034],accel_mss,speed_ms,0,blend_radius_m)
    movel([0.105364, -1.443229, -2.519783, -0.749376, 1.570796, 1.676160],accel_mss,speed_ms,0,blend_radius_m)
    movel([0.103317, -1.444521, -2.518749, -0.749119, 1.570796, 1.674113],accel_mss,speed_ms,0,blend_radius_m)
    movel([0.101180, -1.445533, -2.517936, -0.748919, 1.570796, 1.671977],accel_mss,speed_ms,0,blend_radius_m)
    movel([0.099050, -1.446312, -2.517311, -0.748766, 1.570796, 1.669846],accel_mss,speed_ms,0,blend_radius_m)
    movel([0.093795, -1.447697, -2.516195, -0.748497, 1.570796, 1.664592],accel_mss,speed_ms,0,blend_radius_m)
    movel([0.088839, -1.449042, -2.515109, -0.748238, 1.570796, 1.659636],accel_mss,speed_ms,0,blend_radius_m)
    movel([0.086906, -1.449752, -2.514535, -0.748103, 1.570796, 1.657703],accel_mss,speed_ms,0,blend_radius_m)
    movel([0.085004, -1.450661, -2.513798, -0.747930, 1.570796, 1.655801],accel_mss,speed_ms,0,blend_radius_m)
    movel([0.083219, -1.451795, -2.512877, -0.747717, 1.570796, 1.654015],accel_mss,speed_ms,0,blend_radius_m)
    movel([0.081643, -1.453180, -2.511750, -0.747459, 1.570796, 1.652439],accel_mss,speed_ms,0,blend_radius_m)
    movel([0.082284, -1.453594, -2.511413, -0.747383, 1.570796, 1.653080],accel_mss,speed_ms,0,blend_radius_m)
    movel([0.084167, -1.454631, -2.510566, -0.747192, 1.570796, 1.654964],accel_mss,speed_ms,0,blend_radius_m)
    movel([0.086036, -1.455322, -2.510001, -0.747066, 1.570796, 1.656832],accel_mss,speed_ms,0,blend_radius_m)
    movel([0.087890, -1.455663, -2.509722, -0.747004, 1.570796, 1.658686],accel_mss,speed_ms,0,blend_radius_m)
    movel([0.089734, -1.455653, -2.509730, -0.747006, 1.570796, 1.660530],accel_mss,speed_ms,0,blend_radius_m)
    movel([0.091546, -1.455337, -2.509989, -0.747063, 1.570796, 1.662343],accel_mss,speed_ms,0,blend_radius_m)
    movel([0.093297, -1.454760, -2.510461, -0.747169, 1.570796, 1.664093],accel_mss,speed_ms,0,blend_radius_m)
    movel([0.094994, -1.453918, -2.511148, -0.747323, 1.570796, 1.665790],accel_mss,speed_ms,0,blend_radius_m)
    movel([0.096635, -1.452811, -2.512050, -0.747527, 1.570796, 1.667431],accel_mss,speed_ms,0,blend_radius_m)
    movel([0.089860, -1.459642, -2.506452, -0.746295, 1.570796, 1.660656],accel_mss,speed_ms,0,blend_radius_m)
    movel([0.072686, -1.448648, -2.515427, -0.748314, 1.570796, 1.643483],accel_mss,speed_ms,0,blend_radius_m)
    movel([0.073358, -1.447948, -2.515992, -0.748448, 1.570796, 1.644154],accel_mss,speed_ms,0,blend_radius_m)
    speed_ms = 0.003
    movel([0.073358, -1.441837, -2.513195, -0.757357, 1.570796, 1.644154],accel_mss,speed_ms,0,blend_radius_m)
    speed_ms = 0.05
    movel([0.073358, -1.418214, -2.501717, -0.792458, 1.570796, 1.644154],accel_mss,speed_ms,0,blend_radius_m)
    #M_RunCode9
    movel([0.096184, -1.427284, -2.494664, -0.790441, 1.570796, 1.666981],accel_mss,speed_ms,0,blend_radius_m)
    #M_RunCode3
    movel([0.096184, -1.450724, -2.506032, -0.755633, 1.570796, 1.666981],accel_mss,speed_ms,0,blend_radius_m)
    speed_ms = 0.003
    movel([0.096184, -1.456785, -2.508802, -0.746802, 1.570796, 1.666981],accel_mss,speed_ms,0,blend_radius_m)
    speed_ms = 0.02
    movel([0.097593, -1.455702, -2.509690, -0.746997, 1.570796, 1.668389],accel_mss,speed_ms,0,blend_radius_m)
    movel([0.099096, -1.455183, -2.510114, -0.747091, 1.570796, 1.669892],accel_mss,speed_ms,0,blend_radius_m)
    movel([0.100532, -1.455189, -2.510110, -0.747090, 1.570796, 1.671328],accel_mss,speed_ms,0,blend_radius_m)
    movel([0.101729, -1.455682, -2.509706, -0.747001, 1.570796, 1.672526],accel_mss,speed_ms,0,blend_radius_m)
    movel([0.102540, -1.456557, -2.508989, -0.746843, 1.570796, 1.673336],accel_mss,speed_ms,0,blend_radius_m)
    movel([0.102817, -1.457715, -2.508039, -0.746636, 1.570796, 1.673613],accel_mss,speed_ms,0,blend_radius_m)
    movel([0.102487, -1.459024, -2.506961, -0.746404, 1.570796, 1.673284],accel_mss,speed_ms,0,blend_radius_m)
    movel([0.101471, -1.460360, -2.505859, -0.746170, 1.570796, 1.672267],accel_mss,speed_ms,0,blend_radius_m)
    movel([0.100331, -1.461290, -2.505091, -0.746008, 1.570796, 1.671128],accel_mss,speed_ms,0,blend_radius_m)
    movel([0.099242, -1.461825, -2.504647, -0.745916, 1.570796, 1.670039],accel_mss,speed_ms,0,blend_radius_m)
    movel([0.098163, -1.462439, -2.504139, -0.745811, 1.570796, 1.668959],accel_mss,speed_ms,0,blend_radius_m)
    movel([0.097740, -1.463064, -2.503621, -0.745705, 1.570796, 1.668536],accel_mss,speed_ms,0,blend_radius_m)
    movel([0.097656, -1.463757, -2.503045, -0.745587, 1.570796, 1.668452],accel_mss,speed_ms,0,blend_radius_m)
    movel([0.097883, -1.464412, -2.502500, -0.745477, 1.570796, 1.668679],accel_mss,speed_ms,0,blend_radius_m)
    movel([0.098396, -1.464928, -2.502071, -0.745391, 1.570796, 1.669192],accel_mss,speed_ms,0,blend_radius_m)
    movel([0.099307, -1.465375, -2.501698, -0.745316, 1.570796, 1.670104],accel_mss,speed_ms,0,blend_radius_m)
    movel([0.100349, -1.465575, -2.501531, -0.745283, 1.570796, 1.671145],accel_mss,speed_ms,0,blend_radius_m)
    movel([0.101520, -1.465527, -2.501571, -0.745291, 1.570796, 1.672316],accel_mss,speed_ms,0,blend_radius_m)
    movel([0.102826, -1.465229, -2.501820, -0.745340, 1.570796, 1.673622],accel_mss,speed_ms,0,blend_radius_m)
    movel([0.104186, -1.464702, -2.502259, -0.745428, 1.570796, 1.674982],accel_mss,speed_ms,0,blend_radius_m)
    movel([0.105528, -1.463960, -2.502876, -0.745553, 1.570796, 1.676324],accel_mss,speed_ms,0,blend_radius_m)
    movel([0.106851, -1.463005, -2.503669, -0.745715, 1.570796, 1.677647],accel_mss,speed_ms,0,blend_radius_m)
    movel([0.108159, -1.461834, -2.504640, -0.745915, 1.570796, 1.678955],accel_mss,speed_ms,0,blend_radius_m)
    movel([0.109978, -1.459624, -2.506467, -0.746298, 1.570796, 1.680775],accel_mss,speed_ms,0,blend_radius_m)
    movel([0.111097, -1.457268, -2.508406, -0.746715, 1.570796, 1.681894],accel_mss,speed_ms,0,blend_radius_m)
    movel([0.111370, -1.456051, -2.509404, -0.746934, 1.570796, 1.682166],accel_mss,speed_ms,0,blend_radius_m)
    movel([0.111419, -1.454832, -2.510402, -0.747155, 1.570796, 1.682215],accel_mss,speed_ms,0,blend_radius_m)
    movel([0.110851, -1.452380, -2.512401, -0.747608, 1.570796, 1.681647],accel_mss,speed_ms,0,blend_radius_m)
    movel([0.109332, -1.450009, -2.514327, -0.748054, 1.570796, 1.680128],accel_mss,speed_ms,0,blend_radius_m)
    movel([0.106804, -1.447822, -2.516095, -0.748473, 1.570796, 1.677600],accel_mss,speed_ms,0,blend_radius_m)
    movel([0.117518, -1.437224, -2.524559, -0.750606, 1.570796, 1.688314],accel_mss,speed_ms,0,blend_radius_m)
    movel([0.129939, -1.446214, -2.517390, -0.748785, 1.570796, 1.700735],accel_mss,speed_ms,0,blend_radius_m)
    movel([0.122923, -1.452995, -2.511901, -0.747493, 1.570796, 1.693720],accel_mss,speed_ms,0,blend_radius_m)
    movel([0.124124, -1.451038, -2.513492, -0.747859, 1.570796, 1.694920],accel_mss,speed_ms,0,blend_radius_m)
    movel([0.124786, -1.448938, -2.515193, -0.748258, 1.570796, 1.695582],accel_mss,speed_ms,0,blend_radius_m)
    movel([0.124868, -1.446802, -2.516916, -0.748671, 1.570796, 1.695664],accel_mss,speed_ms,0,blend_radius_m)
    movel([0.124338, -1.444736, -2.518577, -0.749076, 1.570796, 1.695134],accel_mss,speed_ms,0,blend_radius_m)
    movel([0.123179, -1.442832, -2.520101, -0.749456, 1.570796, 1.693975],accel_mss,speed_ms,0,blend_radius_m)
    movel([0.121391, -1.441187, -2.521413, -0.749789, 1.570796, 1.692187],accel_mss,speed_ms,0,blend_radius_m)
    movel([0.113466, -1.448957, -2.515177, -0.748254, 1.570796, 1.684263],accel_mss,speed_ms,0,blend_radius_m)
    movel([0.115713, -1.450913, -2.513593, -0.747883, 1.570796, 1.686509],accel_mss,speed_ms,0,blend_radius_m)
    movel([0.117412, -1.453222, -2.511716, -0.747451, 1.570796, 1.688208],accel_mss,speed_ms,0,blend_radius_m)
    movel([0.118379, -1.455789, -2.509619, -0.746981, 1.570796, 1.689175],accel_mss,speed_ms,0,blend_radius_m)
    movel([0.118524, -1.457134, -2.508515, -0.746739, 1.570796, 1.689320],accel_mss,speed_ms,0,blend_radius_m)
    movel([0.118441, -1.458524, -2.507373, -0.746492, 1.570796, 1.689238],accel_mss,speed_ms,0,blend_radius_m)
    movel([0.118097, -1.459926, -2.506218, -0.746245, 1.570796, 1.688893],accel_mss,speed_ms,0,blend_radius_m)
    movel([0.117452, -1.461313, -2.505072, -0.746004, 1.570796, 1.688248],accel_mss,speed_ms,0,blend_radius_m)
    movel([0.116509, -1.462686, -2.503934, -0.745769, 1.570796, 1.687305],accel_mss,speed_ms,0,blend_radius_m)
    movel([0.115268, -1.464045, -2.502805, -0.745539, 1.570796, 1.686064],accel_mss,speed_ms,0,blend_radius_m)
    movel([0.113855, -1.465280, -2.501777, -0.745332, 1.570796, 1.684652],accel_mss,speed_ms,0,blend_radius_m)
    movel([0.112394, -1.466285, -2.500939, -0.745165, 1.570796, 1.683190],accel_mss,speed_ms,0,blend_radius_m)
    movel([0.110882, -1.467060, -2.500292, -0.745038, 1.570796, 1.681679],accel_mss,speed_ms,0,blend_radius_m)
    movel([0.109317, -1.467606, -2.499835, -0.744949, 1.570796, 1.680114],accel_mss,speed_ms,0,blend_radius_m)
    movel([0.106199, -1.468111, -2.499411, -0.744867, 1.570796, 1.676996],accel_mss,speed_ms,0,blend_radius_m)
    movel([0.103209, -1.467898, -2.499590, -0.744901, 1.570796, 1.674005],accel_mss,speed_ms,0,blend_radius_m)
    movel([0.100457, -1.467096, -2.500261, -0.745032, 1.570796, 1.671254],accel_mss,speed_ms,0,blend_radius_m)
    movel([0.098069, -1.465832, -2.501317, -0.745240, 1.570796, 1.668865],accel_mss,speed_ms,0,blend_radius_m)
    movel([0.096712, -1.464684, -2.502274, -0.745431, 1.570796, 1.667508],accel_mss,speed_ms,0,blend_radius_m)
    movel([0.095606, -1.463254, -2.503463, -0.745672, 1.570796, 1.666403],accel_mss,speed_ms,0,blend_radius_m)
    movel([0.094883, -1.461644, -2.504797, -0.745947, 1.570796, 1.665679],accel_mss,speed_ms,0,blend_radius_m)
    movel([0.094684, -1.459957, -2.506192, -0.746240, 1.570796, 1.665481],accel_mss,speed_ms,0,blend_radius_m)
    movel([0.095089, -1.458302, -2.507556, -0.746531, 1.570796, 1.665886],accel_mss,speed_ms,0,blend_radius_m)
    movel([0.096184, -1.456785, -2.508802, -0.746802, 1.570796, 1.666981],accel_mss,speed_ms,0,blend_radius_m)
    speed_ms = 0.003
    movel([0.096184, -1.450724, -2.506032, -0.755633, 1.570796, 1.666981],accel_mss,speed_ms,0,blend_radius_m)
    speed_ms = 0.05
    movel([0.096184, -1.427284, -2.494664, -0.790441, 1.570796, 1.666981],accel_mss,speed_ms,0,blend_radius_m)
    #M_RunCode9
    movel([0.065363, -1.369061, -2.537910, -0.805417, 1.570796, 1.636159],accel_mss,speed_ms,0,blend_radius_m)
    #M_RunCode3
    movel([0.065363, -1.393636, -2.549996, -0.768757, 1.570796, 1.636159],accel_mss,speed_ms,0,blend_radius_m)
    speed_ms = 0.003
    movel([0.065363, -1.400012, -2.552945, -0.759432, 1.570796, 1.636159],accel_mss,speed_ms,0,blend_radius_m)
    speed_ms = 0.02
    movel([0.062779, -1.401414, -2.551912, -0.759062, 1.570796, 1.633576],accel_mss,speed_ms,0,blend_radius_m)
    movel([0.060012, -1.402408, -2.551179, -0.758802, 1.570796, 1.630808],accel_mss,speed_ms,0,blend_radius_m)
    movel([0.057163, -1.403040, -2.550712, -0.758637, 1.570796, 1.627959],accel_mss,speed_ms,0,blend_radius_m)
    movel([0.054336, -1.403351, -2.550482, -0.758556, 1.570796, 1.625132],accel_mss,speed_ms,0,blend_radius_m)
    movel([0.051638, -1.403378, -2.550462, -0.758549, 1.570796, 1.622434],accel_mss,speed_ms,0,blend_radius_m)
    movel([0.051705, -1.400681, -2.552453, -0.759255, 1.570796, 1.622501],accel_mss,speed_ms,0,blend_radius_m)
    movel([0.052593, -1.397500, -2.554788, -0.760101, 1.570796, 1.623390],accel_mss,speed_ms,0,blend_radius_m)
    movel([0.054194, -1.394122, -2.557251, -0.761016, 1.570796, 1.624991],accel_mss,speed_ms,0,blend_radius_m)
    movel([0.056383, -1.390860, -2.559614, -0.761915, 1.570796, 1.627180],accel_mss,speed_ms,0,blend_radius_m)
    movel([0.059042, -1.388022, -2.561657, -0.762710, 1.570796, 1.629838],accel_mss,speed_ms,0,blend_radius_m)
    movel([0.060505, -1.386862, -2.562489, -0.763038, 1.570796, 1.631301],accel_mss,speed_ms,0,blend_radius_m)
    movel([0.062034, -1.385928, -2.563158, -0.763304, 1.570796, 1.632830],accel_mss,speed_ms,0,blend_radius_m)
    movel([0.063614, -1.385260, -2.563635, -0.763495, 1.570796, 1.634411],accel_mss,speed_ms,0,blend_radius_m)
    movel([0.065228, -1.384898, -2.563893, -0.763598, 1.570796, 1.636025],accel_mss,speed_ms,0,blend_radius_m)
    movel([0.066855, -1.384880, -2.563906, -0.763603, 1.570796, 1.637651],accel_mss,speed_ms,0,blend_radius_m)
    movel([0.068475, -1.385252, -2.563640, -0.763497, 1.570796, 1.639272],accel_mss,speed_ms,0,blend_radius_m)
    movel([0.070360, -1.386422, -2.562804, -0.763163, 1.570796, 1.641156],accel_mss,speed_ms,0,blend_radius_m)
    movel([0.071352, -1.388167, -2.561553, -0.762669, 1.570796, 1.642148],accel_mss,speed_ms,0,blend_radius_m)
    movel([0.071524, -1.390371, -2.559967, -0.762051, 1.570796, 1.642320],accel_mss,speed_ms,0,blend_radius_m)
    movel([0.070946, -1.392916, -2.558126, -0.761347, 1.570796, 1.641743],accel_mss,speed_ms,0,blend_radius_m)
    movel([0.069554, -1.395810, -2.556022, -0.760557, 1.570796, 1.640350],accel_mss,speed_ms,0,blend_radius_m)
    movel([0.067656, -1.398159, -2.554305, -0.759925, 1.570796, 1.638453],accel_mss,speed_ms,0,blend_radius_m)
    movel([0.065363, -1.400012, -2.552945, -0.759432, 1.570796, 1.636159],accel_mss,speed_ms,0,blend_radius_m)
    speed_ms = 0.003
    movel([0.065363, -1.393636, -2.549996, -0.768757, 1.570796, 1.636159],accel_mss,speed_ms,0,blend_radius_m)
    speed_ms = 0.05
    movel([0.065363, -1.369061, -2.537910, -0.805417, 1.570796, 1.636159],accel_mss,speed_ms,0,blend_radius_m)
    #M_RunCode9
    movel([0.108201, -1.279960, -2.595203, -0.837226, 1.570796, 1.678998],accel_mss,speed_ms,0,blend_radius_m)
    #M_RunCode3
    movel([0.108201, -1.306030, -2.608435, -0.797923, 1.570796, 1.678998],accel_mss,speed_ms,0,blend_radius_m)
    speed_ms = 0.003
    movel([0.108201, -1.312833, -2.611673, -0.787882, 1.570796, 1.678998],accel_mss,speed_ms,0,blend_radius_m)
    speed_ms = 0.02
    movel([0.106517, -1.312610, -2.611810, -0.787968, 1.570796, 1.677313],accel_mss,speed_ms,0,blend_radius_m)
    movel([0.105092, -1.311943, -2.612220, -0.788226, 1.570796, 1.675888],accel_mss,speed_ms,0,blend_radius_m)
    movel([0.103827, -1.311038, -2.612774, -0.788577, 1.570796, 1.674623],accel_mss,speed_ms,0,blend_radius_m)
    movel([0.104560, -1.310549, -2.613073, -0.788767, 1.570796, 1.675356],accel_mss,speed_ms,0,blend_radius_m)
    movel([0.105215, -1.310555, -2.613069, -0.788765, 1.570796, 1.676012],accel_mss,speed_ms,0,blend_radius_m)
    movel([0.105997, -1.310511, -2.613096, -0.788782, 1.570796, 1.676793],accel_mss,speed_ms,0,blend_radius_m)
    movel([0.107100, -1.309876, -2.613484, -0.789029, 1.570796, 1.677896],accel_mss,speed_ms,0,blend_radius_m)
    movel([0.108084, -1.308861, -2.614103, -0.789425, 1.570796, 1.678880],accel_mss,speed_ms,0,blend_radius_m)
    movel([0.108901, -1.307727, -2.614792, -0.789870, 1.570796, 1.679697],accel_mss,speed_ms,0,blend_radius_m)
    movel([0.109984, -1.306129, -2.615761, -0.790499, 1.570796, 1.680780],accel_mss,speed_ms,0,blend_radius_m)
    movel([0.108500, -1.304879, -2.616517, -0.790993, 1.570796, 1.679297],accel_mss,speed_ms,0,blend_radius_m)
    movel([0.106768, -1.304387, -2.616814, -0.791188, 1.570796, 1.677564],accel_mss,speed_ms,0,blend_radius_m)
    movel([0.105805, -1.304516, -2.616736, -0.791137, 1.570796, 1.676602],accel_mss,speed_ms,0,blend_radius_m)
    movel([0.104779, -1.304946, -2.616477, -0.790967, 1.570796, 1.675575],accel_mss,speed_ms,0,blend_radius_m)
    movel([0.103687, -1.305712, -2.616013, -0.790663, 1.570796, 1.674483],accel_mss,speed_ms,0,blend_radius_m)
    movel([0.102532, -1.306852, -2.615323, -0.790214, 1.570796, 1.673328],accel_mss,speed_ms,0,blend_radius_m)
    movel([0.102352, -1.305645, -2.616054, -0.790690, 1.570796, 1.673149],accel_mss,speed_ms,0,blend_radius_m)
    movel([0.102385, -1.304530, -2.616728, -0.791132, 1.570796, 1.673181],accel_mss,speed_ms,0,blend_radius_m)
    movel([0.102578, -1.304058, -2.617012, -0.791319, 1.570796, 1.673375],accel_mss,speed_ms,0,blend_radius_m)
    movel([0.102946, -1.303674, -2.617244, -0.791472, 1.570796, 1.673743],accel_mss,speed_ms,0,blend_radius_m)
    movel([0.104357, -1.303249, -2.617500, -0.791641, 1.570796, 1.675154],accel_mss,speed_ms,0,blend_radius_m)
    movel([0.107054, -1.303315, -2.617459, -0.791614, 1.570796, 1.677851],accel_mss,speed_ms,0,blend_radius_m)
    movel([0.109447, -1.304023, -2.617034, -0.791333, 1.570796, 1.680243],accel_mss,speed_ms,0,blend_radius_m)
    movel([0.110353, -1.304653, -2.616653, -0.791083, 1.570796, 1.681150],accel_mss,speed_ms,0,blend_radius_m)
    movel([0.110971, -1.305491, -2.616147, -0.790751, 1.570796, 1.681767],accel_mss,speed_ms,0,blend_radius_m)
    movel([0.111233, -1.306548, -2.615508, -0.790334, 1.570796, 1.682029],accel_mss,speed_ms,0,blend_radius_m)
    movel([0.111068, -1.307839, -2.614724, -0.789826, 1.570796, 1.681865],accel_mss,speed_ms,0,blend_radius_m)
    movel([0.109348, -1.307847, -2.614720, -0.789823, 1.570796, 1.680145],accel_mss,speed_ms,0,blend_radius_m)
    movel([0.110243, -1.312399, -2.611940, -0.788050, 1.570796, 1.681040],accel_mss,speed_ms,0,blend_radius_m)
    movel([0.108201, -1.312833, -2.611673, -0.787882, 1.570796, 1.678998],accel_mss,speed_ms,0,blend_radius_m)
    speed_ms = 0.003
    movel([0.108201, -1.306030, -2.608435, -0.797923, 1.570796, 1.678998],accel_mss,speed_ms,0,blend_radius_m)
    speed_ms = 0.05
    movel([0.108201, -1.279960, -2.595203, -0.837226, 1.570796, 1.678998],accel_mss,speed_ms,0,blend_radius_m)
    #M_RunCode9
    movel([0.068183, -1.263928, -2.604442, -0.844019, 1.570796, 1.638979],accel_mss,speed_ms,0,blend_radius_m)
    #M_RunCode3
    movel([0.068183, -1.290226, -2.617885, -0.804278, 1.570796, 1.638979],accel_mss,speed_ms,0,blend_radius_m)
    speed_ms = 0.003
    movel([0.068183, -1.297097, -2.621176, -0.794116, 1.570796, 1.638979],accel_mss,speed_ms,0,blend_radius_m)
    speed_ms = 0.02
    movel([0.066467, -1.299361, -2.619829, -0.793200, 1.570796, 1.637264],accel_mss,speed_ms,0,blend_radius_m)
    movel([0.064519, -1.301543, -2.618524, -0.792322, 1.570796, 1.635316],accel_mss,speed_ms,0,blend_radius_m)
    movel([0.062350, -1.303607, -2.617284, -0.791498, 1.570796, 1.633146],accel_mss,speed_ms,0,blend_radius_m)
    movel([0.059974, -1.305526, -2.616126, -0.790737, 1.570796, 1.630771],accel_mss,speed_ms,0,blend_radius_m)
    movel([0.057413, -1.307268, -2.615071, -0.790050, 1.570796, 1.628210],accel_mss,speed_ms,0,blend_radius_m)
    movel([0.055975, -1.307970, -2.614644, -0.789774, 1.570796, 1.626771],accel_mss,speed_ms,0,blend_radius_m)
    movel([0.054432, -1.308529, -2.614305, -0.789555, 1.570796, 1.625229],accel_mss,speed_ms,0,blend_radius_m)
    movel([0.053046, -1.309040, -2.613993, -0.789355, 1.570796, 1.623842],accel_mss,speed_ms,0,blend_radius_m)
    movel([0.052086, -1.309587, -2.613660, -0.789142, 1.570796, 1.622882],accel_mss,speed_ms,0,blend_radius_m)
    movel([0.050909, -1.311045, -2.612770, -0.788574, 1.570796, 1.621705],accel_mss,speed_ms,0,blend_radius_m)
    movel([0.049542, -1.313173, -2.611465, -0.787751, 1.570796, 1.620338],accel_mss,speed_ms,0,blend_radius_m)
    movel([0.048143, -1.315401, -2.610092, -0.786896, 1.570796, 1.618940],accel_mss,speed_ms,0,blend_radius_m)
    movel([0.046861, -1.317165, -2.609001, -0.786223, 1.570796, 1.617657],accel_mss,speed_ms,0,blend_radius_m)
    movel([0.043920, -1.320192, -2.607119, -0.785078, 1.570796, 1.614716],accel_mss,speed_ms,0,blend_radius_m)
    movel([0.041006, -1.322557, -2.605639, -0.784192, 1.570796, 1.611803],accel_mss,speed_ms,0,blend_radius_m)
    movel([0.038118, -1.324329, -2.604527, -0.783534, 1.570796, 1.608914],accel_mss,speed_ms,0,blend_radius_m)
    movel([0.035257, -1.325566, -2.603747, -0.783076, 1.570796, 1.606054],accel_mss,speed_ms,0,blend_radius_m)
    movel([0.032430, -1.326331, -2.603264, -0.782794, 1.570796, 1.603226],accel_mss,speed_ms,0,blend_radius_m)
    movel([0.029639, -1.326680, -2.603043, -0.782666, 1.570796, 1.600436],accel_mss,speed_ms,0,blend_radius_m)
    movel([0.026891, -1.326669, -2.603050, -0.782670, 1.570796, 1.597687],accel_mss,speed_ms,0,blend_radius_m)
    movel([0.024187, -1.326357, -2.603248, -0.782785, 1.570796, 1.594984],accel_mss,speed_ms,0,blend_radius_m)
    movel([0.018950, -1.325045, -2.604075, -0.783268, 1.570796, 1.589746],accel_mss,speed_ms,0,blend_radius_m)
    movel([0.013993, -1.323179, -2.605249, -0.783961, 1.570796, 1.584790],accel_mss,speed_ms,0,blend_radius_m)
    movel([0.005237, -1.319507, -2.607546, -0.785336, 1.570796, 1.576034],accel_mss,speed_ms,0,blend_radius_m)
    movel([0.001064, -1.318336, -2.608275, -0.785779, 1.570796, 1.571861],accel_mss,speed_ms,0,blend_radius_m)
    movel([-0.004062, -1.317433, -2.608835, -0.786121, 1.570796, 1.566734],accel_mss,speed_ms,0,blend_radius_m)
    movel([-0.009890, -1.316882, -2.609177, -0.786331, 1.570796, 1.560907],accel_mss,speed_ms,0,blend_radius_m)
    movel([-0.016155, -1.316757, -2.609254, -0.786378, 1.570796, 1.554641],accel_mss,speed_ms,0,blend_radius_m)
    movel([-0.022589, -1.317129, -2.609023, -0.786237, 1.570796, 1.548207],accel_mss,speed_ms,0,blend_radius_m)
    movel([-0.028918, -1.318053, -2.608450, -0.785886, 1.570796, 1.541878],accel_mss,speed_ms,0,blend_radius_m)
    movel([-0.034863, -1.319579, -2.607501, -0.785309, 1.570796, 1.535934],accel_mss,speed_ms,0,blend_radius_m)
    movel([-0.037604, -1.320583, -2.606874, -0.784931, 1.570796, 1.533193],accel_mss,speed_ms,0,blend_radius_m)
    movel([-0.040145, -1.321751, -2.606144, -0.784493, 1.570796, 1.530652],accel_mss,speed_ms,0,blend_radius_m)
    movel([-0.042700, -1.323193, -2.605240, -0.783955, 1.570796, 1.528096],accel_mss,speed_ms,0,blend_radius_m)
    movel([-0.045606, -1.325084, -2.604051, -0.783254, 1.570796, 1.525190],accel_mss,speed_ms,0,blend_radius_m)
    movel([-0.048654, -1.327357, -2.602615, -0.782417, 1.570796, 1.522142],accel_mss,speed_ms,0,blend_radius_m)
    movel([-0.051646, -1.329942, -2.600973, -0.781474, 1.570796, 1.519150],accel_mss,speed_ms,0,blend_radius_m)
    movel([-0.054374, -1.332764, -2.599170, -0.780455, 1.570796, 1.516423],accel_mss,speed_ms,0,blend_radius_m)
    movel([-0.056644, -1.335756, -2.597247, -0.779386, 1.570796, 1.514152],accel_mss,speed_ms,0,blend_radius_m)
    movel([-0.058260, -1.338847, -2.595248, -0.778294, 1.570796, 1.512537],accel_mss,speed_ms,0,blend_radius_m)
    movel([-0.058764, -1.340407, -2.594234, -0.777748, 1.570796, 1.512032],accel_mss,speed_ms,0,blend_radius_m)
    movel([-0.059032, -1.341968, -2.593216, -0.777205, 1.570796, 1.511764],accel_mss,speed_ms,0,blend_radius_m)
    movel([-0.058880, -1.344184, -2.591765, -0.776440, 1.570796, 1.511916],accel_mss,speed_ms,0,blend_radius_m)
    movel([-0.058008, -1.345772, -2.590721, -0.775896, 1.570796, 1.512788],accel_mss,speed_ms,0,blend_radius_m)
    movel([-0.056501, -1.346799, -2.590044, -0.775545, 1.570796, 1.514295],accel_mss,speed_ms,0,blend_radius_m)
    movel([-0.054442, -1.347330, -2.589694, -0.775365, 1.570796, 1.516354],accel_mss,speed_ms,0,blend_radius_m)
    movel([-0.051910, -1.347426, -2.589630, -0.775332, 1.570796, 1.518886],accel_mss,speed_ms,0,blend_radius_m)
    movel([-0.048987, -1.347151, -2.589812, -0.775426, 1.570796, 1.521810],accel_mss,speed_ms,0,blend_radius_m)
    movel([-0.045747, -1.346563, -2.590200, -0.775626, 1.570796, 1.525049],accel_mss,speed_ms,0,blend_radius_m)
    movel([-0.042271, -1.345725, -2.590752, -0.775912, 1.570796, 1.528526],accel_mss,speed_ms,0,blend_radius_m)
    movel([-0.034933, -1.343530, -2.592194, -0.776665, 1.570796, 1.535863],accel_mss,speed_ms,0,blend_radius_m)
    movel([-0.027609, -1.341035, -2.593825, -0.777529, 1.570796, 1.543188],accel_mss,speed_ms,0,blend_radius_m)
    movel([-0.020959, -1.338699, -2.595344, -0.778346, 1.570796, 1.549838],accel_mss,speed_ms,0,blend_radius_m)
    movel([-0.015651, -1.336987, -2.596453, -0.778949, 1.570796, 1.555145],accel_mss,speed_ms,0,blend_radius_m)
    movel([-0.002809, -1.333318, -2.598815, -0.780256, 1.570796, 1.567988],accel_mss,speed_ms,0,blend_radius_m)
    movel([0.004059, -1.331537, -2.599955, -0.780897, 1.570796, 1.574855],accel_mss,speed_ms,0,blend_radius_m)
    movel([0.009383, -1.330453, -2.600647, -0.781289, 1.570796, 1.580179],accel_mss,speed_ms,0,blend_radius_m)
    movel([0.011398, -1.330291, -2.600751, -0.781348, 1.570796, 1.582194],accel_mss,speed_ms,0,blend_radius_m)
    movel([0.013270, -1.330370, -2.600700, -0.781319, 1.570796, 1.584066],accel_mss,speed_ms,0,blend_radius_m)
    movel([0.016577, -1.331200, -2.600171, -0.781018, 1.570796, 1.587373],accel_mss,speed_ms,0,blend_radius_m)
    movel([0.019297, -1.332810, -2.599141, -0.780438, 1.570796, 1.590093],accel_mss,speed_ms,0,blend_radius_m)
    movel([0.021435, -1.335056, -2.597698, -0.779635, 1.570796, 1.592231],accel_mss,speed_ms,0,blend_radius_m)
    movel([0.022985, -1.337804, -2.595924, -0.778661, 1.570796, 1.593781],accel_mss,speed_ms,0,blend_radius_m)
    movel([0.023955, -1.340917, -2.593902, -0.777570, 1.570796, 1.594751],accel_mss,speed_ms,0,blend_radius_m)
    movel([0.024352, -1.344258, -2.591716, -0.776414, 1.570796, 1.595148],accel_mss,speed_ms,0,blend_radius_m)
    movel([0.024181, -1.347692, -2.589455, -0.775242, 1.570796, 1.594978],accel_mss,speed_ms,0,blend_radius_m)
    movel([0.023212, -1.352030, -2.586574, -0.773785, 1.570796, 1.594008],accel_mss,speed_ms,0,blend_radius_m)
    movel([0.022491, -1.353877, -2.585340, -0.773172, 1.570796, 1.593287],accel_mss,speed_ms,0,blend_radius_m)
    movel([0.021617, -1.355544, -2.584222, -0.772623, 1.570796, 1.592413],accel_mss,speed_ms,0,blend_radius_m)
    movel([0.020604, -1.357053, -2.583206, -0.772130, 1.570796, 1.591400],accel_mss,speed_ms,0,blend_radius_m)
    movel([0.019454, -1.358428, -2.582278, -0.771683, 1.570796, 1.590251],accel_mss,speed_ms,0,blend_radius_m)
    movel([0.016782, -1.360879, -2.580617, -0.770893, 1.570796, 1.587578],accel_mss,speed_ms,0,blend_radius_m)
    movel([0.013656, -1.363086, -2.579115, -0.770188, 1.570796, 1.584452],accel_mss,speed_ms,0,blend_radius_m)
    movel([0.010137, -1.365236, -2.577644, -0.769509, 1.570796, 1.580933],accel_mss,speed_ms,0,blend_radius_m)
    movel([0.002163, -1.370091, -2.574300, -0.767998, 1.570796, 1.572959],accel_mss,speed_ms,0,blend_radius_m)
    movel([0.001770, -1.370367, -2.574108, -0.767913, 1.570796, 1.572566],accel_mss,speed_ms,0,blend_radius_m)
    movel([0.001962, -1.370367, -2.574109, -0.767914, 1.570796, 1.572759],accel_mss,speed_ms,0,blend_radius_m)
    movel([0.003797, -1.369678, -2.574586, -0.768126, 1.570796, 1.574594],accel_mss,speed_ms,0,blend_radius_m)
    movel([0.011160, -1.366566, -2.576731, -0.769092, 1.570796, 1.581956],accel_mss,speed_ms,0,blend_radius_m)
    movel([0.023447, -1.361411, -2.580256, -0.770722, 1.570796, 1.594243],accel_mss,speed_ms,0,blend_radius_m)
    movel([0.017685, -1.366383, -2.576857, -0.769149, 1.570796, 1.588482],accel_mss,speed_ms,0,blend_radius_m)
    movel([0.011119, -1.371663, -2.573210, -0.767516, 1.570796, 1.581916],accel_mss,speed_ms,0,blend_radius_m)
    movel([0.004025, -1.377088, -2.569421, -0.765880, 1.570796, 1.574821],accel_mss,speed_ms,0,blend_radius_m)
    movel([-0.003343, -1.382493, -2.565605, -0.764291, 1.570796, 1.567454],accel_mss,speed_ms,0,blend_radius_m)
    movel([-0.017889, -1.392616, -2.558343, -0.761429, 1.570796, 1.552908],accel_mss,speed_ms,0,blend_radius_m)
    movel([-0.024590, -1.397017, -2.555141, -0.760231, 1.570796, 1.546206],accel_mss,speed_ms,0,blend_radius_m)
    movel([-0.030606, -1.400773, -2.552385, -0.759231, 1.570796, 1.540190],accel_mss,speed_ms,0,blend_radius_m)
    movel([-0.037332, -1.408268, -2.546824, -0.757297, 1.570796, 1.533464],accel_mss,speed_ms,0,blend_radius_m)
    movel([-0.043886, -1.416131, -2.540902, -0.755356, 1.570796, 1.526910],accel_mss,speed_ms,0,blend_radius_m)
    movel([-0.056627, -1.432235, -2.528484, -0.751670, 1.570796, 1.514169],accel_mss,speed_ms,0,blend_radius_m)
    movel([-0.062904, -1.440143, -2.522245, -0.750002, 1.570796, 1.507892],accel_mss,speed_ms,0,blend_radius_m)
    movel([-0.069187, -1.447749, -2.516153, -0.748487, 1.570796, 1.501610],accel_mss,speed_ms,0,blend_radius_m)
    movel([-0.075526, -1.454908, -2.510340, -0.747142, 1.570796, 1.495270],accel_mss,speed_ms,0,blend_radius_m)
    movel([-0.081984, -1.461480, -2.504933, -0.745976, 1.570796, 1.488813],accel_mss,speed_ms,0,blend_radius_m)
    movel([-0.084611, -1.463841, -2.502975, -0.745573, 1.570796, 1.486186],accel_mss,speed_ms,0,blend_radius_m)
    movel([-0.087222, -1.465905, -2.501256, -0.745228, 1.570796, 1.483574],accel_mss,speed_ms,0,blend_radius_m)
    movel([-0.089796, -1.467667, -2.499783, -0.744939, 1.570796, 1.481000],accel_mss,speed_ms,0,blend_radius_m)
    movel([-0.092315, -1.469128, -2.498559, -0.744703, 1.570796, 1.478481],accel_mss,speed_ms,0,blend_radius_m)
    movel([-0.094761, -1.470280, -2.497591, -0.744519, 1.570796, 1.476035],accel_mss,speed_ms,0,blend_radius_m)
    movel([-0.097118, -1.471120, -2.496884, -0.744386, 1.570796, 1.473678],accel_mss,speed_ms,0,blend_radius_m)
    movel([-0.099367, -1.471645, -2.496441, -0.744303, 1.570796, 1.471430],accel_mss,speed_ms,0,blend_radius_m)
    movel([-0.101485, -1.471850, -2.496268, -0.744271, 1.570796, 1.469311],accel_mss,speed_ms,0,blend_radius_m)
    movel([-0.103458, -1.471728, -2.496371, -0.744290, 1.570796, 1.467338],accel_mss,speed_ms,0,blend_radius_m)
    movel([-0.105267, -1.471271, -2.496756, -0.744362, 1.570796, 1.465529],accel_mss,speed_ms,0,blend_radius_m)
    movel([-0.106888, -1.470476, -2.497426, -0.744487, 1.570796, 1.463908],accel_mss,speed_ms,0,blend_radius_m)
    movel([-0.108306, -1.469335, -2.498385, -0.744669, 1.570796, 1.462490],accel_mss,speed_ms,0,blend_radius_m)
    movel([-0.109498, -1.467837, -2.499641, -0.744911, 1.570796, 1.461298],accel_mss,speed_ms,0,blend_radius_m)
    movel([-0.110443, -1.465975, -2.501198, -0.745216, 1.570796, 1.460354],accel_mss,speed_ms,0,blend_radius_m)
    movel([-0.111118, -1.463738, -2.503060, -0.745590, 1.570796, 1.459678],accel_mss,speed_ms,0,blend_radius_m)
    movel([-0.111501, -1.461116, -2.505234, -0.746038, 1.570796, 1.459295],accel_mss,speed_ms,0,blend_radius_m)
    movel([-0.108428, -1.460890, -2.505421, -0.746077, 1.570796, 1.462368],accel_mss,speed_ms,0,blend_radius_m)
    movel([-0.106908, -1.460703, -2.505576, -0.746110, 1.570796, 1.463888],accel_mss,speed_ms,0,blend_radius_m)
    movel([-0.105411, -1.460222, -2.505973, -0.746194, 1.570796, 1.465385],accel_mss,speed_ms,0,blend_radius_m)
    movel([-0.104290, -1.459531, -2.506543, -0.746314, 1.570796, 1.466507],accel_mss,speed_ms,0,blend_radius_m)
    movel([-0.103032, -1.458465, -2.507421, -0.746502, 1.570796, 1.467764],accel_mss,speed_ms,0,blend_radius_m)
    movel([-0.100191, -1.455393, -2.509943, -0.747053, 1.570796, 1.470605],accel_mss,speed_ms,0,blend_radius_m)
